KUKA KRL program: MyProgram_327().src

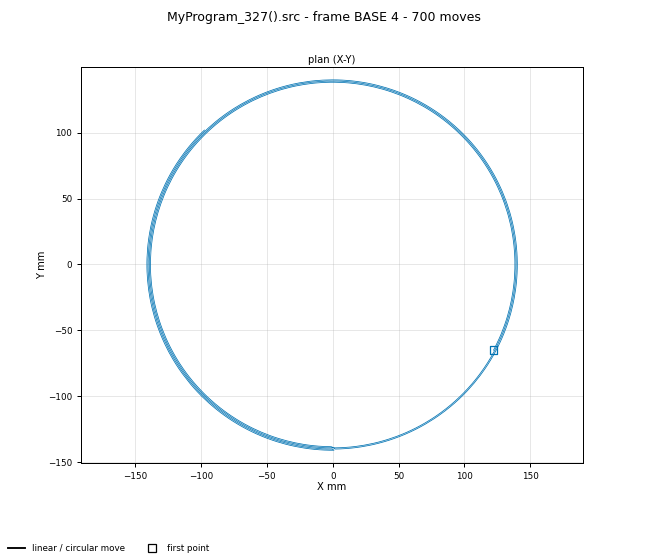
[picture p0: tool path of MyProgram_327().src in frame BASE 4, 700 of 700 moves have a stored position in this frame; points joined in program order, loops and branches not executed]
&ACCESS RVP
&REL 1
&PARAM TEMPLATE = C:\KRC\Roboter\Template\vorgabe
&PARAM EDITMASK = *
DEF MyProgram_327()
; ---- Setting reference (Base) ----
$BASE = BASE_DATA[4]

; --------------------------
; ---- Setting tool (TCP) ----
$TOOL = TOOL_DATA[3]
; --------------------------

$VEL.CP = VEL_APROX_PRINT
Startdeposition()
$VEL.CP = VEL_PRINT
LIN {X 122.1001,Y -65.1036,Z 187,A -22.8126,B 2.4164,C 0.2067,E1 2.5678,E2 476.0313} C_DIS
LIN {X 123.7198,Y -61.9701,Z 187,A -21.3071,B 2.4167,C 0.2026,E1 2.5697,E2 474.5187} C_DIS
LIN {X 125.4053,Y -58.4798,Z 187,A -19.8742,B 2.417,C 0.2,E1 2.5714,E2 473.1074} C_DIS
LIN {X 126.6756,Y -55.679,Z 187,A -18.6979,B 2.4172,C 0.1975,E1 2.5727,E2 471.9431} C_DIS
LIN {X 128.0646,Y -52.404,Z 187,A -17.2,B 2.4175,C 0.1934,E1 2.5743,E2 470.4408} C_DIS
LIN {X 129.3229,Y -49.2171,Z 187,A -15.9923,B 2.4177,C 0.1914,E1 2.5755,E2 469.2602} C_DIS
LIN {X 130.4667,Y -46.1012,Z 187,A -14.659,B 2.4179,C 0.1881,E1 2.5768,E2 467.9313} C_DIS
LIN {X 131.5504,Y -42.9116,Z 187,A -13.3395,B 2.4182,C 0.185,E1 2.5779,E2 466.6208} C_DIS
LIN {X 132.6605,Y -39.3399,Z 187,A -11.9013,B 2.4184,C 0.1818,E1 2.5791,E2 465.1961} C_DIS
LIN {X 133.607,Y -35.9933,Z 187,A -10.6668,B 2.4186,C 0.1796,E1 2.58,E2 463.9876} C_DIS
LIN {X 134.3292,Y -33.2047,Z 187,A -9.3124,B 2.4189,C 0.175,E1 2.5809,E2 462.6111} C_DIS
LIN {X 135.0798,Y -30.0064,Z 187,A -8.0933,B 2.4191,C 0.1724,E1 2.5817,E2 461.4097} C_DIS
LIN {X 135.7603,Y -26.7586,Z 187,A -6.8145,B 2.4193,C 0.1695,E1 2.5824,E2 460.1425} C_DIS
LIN {X 136.44,Y -23.0315,Z 187,A -5.513,B 2.4194,C 0.1674,E1 2.583,E2 458.875} C_DIS
LIN {X 136.8645,Y -20.3723,Z 187,A -4.2723,B 2.4197,C 0.1632,E1 2.5835,E2 457.6172} C_DIS
LIN {X 137.3012,Y -17.1844,Z 187,A -3.0154,B 2.4199,C 0.1602,E1 2.584,E2 456.3692} C_DIS
LIN {X 137.6611,Y -14.0125,Z 187,A -1.7682,B 2.4201,C 0.1571,E1 2.5844,E2 455.1309} C_DIS
LIN {X 137.9882,Y -10.2764,Z 187,A -0.3069,B 2.4204,C 0.1535,E1 2.5847,E2 453.6806} C_DIS
LIN {X 138.2359,Y -6.1423,Z 187,A 1.3133,B 2.4206,C 0.1495,E1 2.5849,E2 452.0716} C_DIS
LIN {X 138.3383,Y -3.0713,Z 187,A 2.5305,B 2.4208,C 0.1464,E1 2.585,E2 450.8609} C_DIS
LIN {X 138.3721,Y 0,Z 187,A 3.7049,B 2.421,C 0.1437,E1 2.585,E2 449.6983} C_DIS
LIN {X 138.3383,Y 3.0713,Z 187,A 5.0506,B 2.4212,C 0.1395,E1 2.585,E2 448.3422} C_DIS
LIN {X 138.1565,Y 7.7265,Z 187,A 6.7524,B 2.4214,C 0.136,E1 2.5847,E2 446.6689} C_DIS
LIN {X 137.9434,Y 10.8859,Z 187,A 8.0939,B 2.4216,C 0.1321,E1 2.5845,E2 445.3227} C_DIS
LIN {X 137.6582,Y 14.0395,Z 187,A 9.2261,B 2.4217,C 0.13,E1 2.5842,E2 444.213} C_DIS
LIN {X 137.2977,Y 17.2115,Z 187,A 10.4775,B 2.4219,C 0.1269,E1 2.5838,E2 442.97} C_DIS
LIN {X 136.8603,Y 20.3995,Z 187,A 11.7392,B 2.4221,C 0.1238,E1 2.5833,E2 441.7166} C_DIS
LIN {X 136.3447,Y 23.601,Z 187,A 13.0011,B 2.4222,C 0.1207,E1 2.5827,E2 440.4644} C_DIS
LIN {X 135.7551,Y 26.786,Z 187,A 14.2905,B 2.4224,C 0.1175,E1 2.582,E2 439.181} C_DIS
LIN {X 135.0798,Y 30.0064,Z 187,A 15.6961,B 2.4226,C 0.1134,E1 2.5812,E2 437.7692} C_DIS
LIN {X 134.1907,Y 33.7517,Z 187,A 17.0979,B 2.4227,C 0.1106,E1 2.5802,E2 436.3913} C_DIS
LIN {X 133.4748,Y 36.4878,Z 187,A 18.1916,B 2.4228,C 0.1081,E1 2.5795,E2 435.307} C_DIS
LIN {X 132.5503,Y 39.7152,Z 187,A 19.5791,B 2.423,C 0.1043,E1 2.5784,E2 433.9191} C_DIS
LIN {X 131.4456,Y 43.2265,Z 187,A 20.9447,B 2.423,C 0.1016,E1 2.5772,E2 432.5732} C_DIS
LIN {X 130.366,Y 46.3814,Z 187,A 22.1708,B 2.4232,C 0.0992,E1 2.5761,E2 431.3662} C_DIS
LIN {X 129.2679,Y 49.3627,Z 187,A 23.5123,B 2.4233,C 0.0955,E1 2.5748,E2 430.0209} C_DIS
LIN {X 127.8426,Y 52.9399,Z 187,A 25.0213,B 2.4235,C 0.092,E1 2.5732,E2 428.522} C_DIS
LIN {X 126.4516,Y 56.1808,Z 187,A 26.2465,B 2.4235,C 0.0902,E1 2.5719,E2 427.3262} C_DIS
LIN {X 125.2281,Y 58.863,Z 187,A 27.5721,B 2.4237,C 0.0861,E1 2.5703,E2 425.9869} C_DIS
LIN {X 123.6932,Y 62.0232,Z 187,A 29.0699,B 2.4238,C 0.0821,E1 2.5684,E2 424.4831} C_DIS
LIN {X 121.6853,Y 65.8758,Z 187,A 30.6655,B 2.4239,C 0.0792,E1 2.5664,E2 422.9127} C_DIS
LIN {X 119.9657,Y 68.9575,Z 187,A 32.0559,B 2.424,C 0.0762,E1 2.5645,E2 421.5308} C_DIS
LIN {X 117.854,Y 72.5066,Z 187,A 33.7517,B 2.4242,C 0.0721,E1 2.562,E2 419.8363} C_DIS
LIN {X 115.8171,Y 75.7187,Z 187,A 35.1883,B 2.4242,C 0.0694,E1 2.5599,E2 418.4167} C_DIS
LIN {X 113.8287,Y 78.6762,Z 187,A 36.5912,B 2.4243,C 0.0665,E1 2.5577,E2 417.0225} C_DIS
LIN {X 111.4897,Y 81.9559,Z 187,A 38.2376,B 2.4244,C 0.0628,E1 2.555,E2 415.3784} C_DIS
LIN {X 109.0842,Y 85.1325,Z 187,A 39.7581,B 2.4244,C 0.06,E1 2.5524,E2 413.8739} C_DIS
LIN {X 106.8509,Y 87.9193,Z 187,A 41.1713,B 2.4245,C 0.0572,E1 2.55,E2 412.4686} C_DIS
LIN {X 104.2126,Y 91.03,Z 187,A 42.8402,B 2.4246,C 0.0537,E1 2.5469,E2 410.8019} C_DIS
LIN {X 101.5684,Y 93.9722,Z 187,A 44.3542,B 2.4246,C 0.0511,E1 2.5441,E2 409.3031} C_DIS
LIN {X 98.7051,Y 96.9744,Z 187,A 46.0508,B 2.4248,C 0.0477,E1 2.5408,E2 407.6089} C_DIS
LIN {X 95.915,Y 99.7357,Z 187,A 47.5589,B 2.4248,C 0.0452,E1 2.5378,E2 406.1153} C_DIS
LIN {X 93.3132,Y 102.1742,Z 187,A 48.9762,B 2.4248,C 0.0427,E1 2.5349,E2 404.7052} C_DIS
LIN {X 90.2523,Y 104.8869,Z 187,A 50.655,B 2.4249,C 0.0396,E1 2.5314,E2 403.0281} C_DIS
LIN {X 87.2159,Y 107.4259,Z 187,A 52.1798,B 2.4249,C 0.0373,E1 2.5281,E2 401.5174} C_DIS
LIN {X 83.9895,Y 109.9659,Z 187,A 53.8641,B 2.4249,C 0.0344,E1 2.5244,E2 399.835} C_DIS
LIN {X 80.6649,Y 112.4275,Z 187,A 55.4338,B 2.425,C 0.0324,E1 2.5209,E2 398.283} C_DIS
LIN {X 77.9316,Y 114.3398,Z 187,A 56.8056,B 2.425,C 0.0301,E1 2.5177,E2 396.9124} C_DIS
LIN {X 74.9631,Y 116.3075,Z 187,A 58.222,B 2.425,C 0.0281,E1 2.5144,E2 395.5032} C_DIS
LIN {X 71.9662,Y 118.1854,Z 187,A 59.6383,B 2.425,C 0.0261,E1 2.5111,E2 394.0929} C_DIS
LIN {X 68.9446,Y 119.9732,Z 187,A 61.0497,B 2.4251,C 0.0241,E1 2.5077,E2 392.6868} C_DIS
LIN {X 65.8626,Y 121.6923,Z 187,A 62.5626,B 2.4251,C 0.0216,E1 2.504,E2 391.1677} C_DIS
LIN {X 63.1849,Y 123.1018,Z 187,A 63.5476,B 2.4251,C 0.0216,E1 2.5016,E2 390.2156} C_DIS
LIN {X 60.4063,Y 124.4908,Z 187,A 64.9206,B 2.4251,C 0.0193,E1 2.4981,E2 388.8323} C_DIS
LIN {X 57.2872,Y 125.9567,Z 187,A 66.4596,B 2.4251,C 0.0167,E1 2.4942,E2 387.2797} C_DIS
LIN {X 54.0928,Y 127.3611,Z 187,A 67.7144,B 2.4251,C 0.0162,E1 2.491,E2 386.0484} C_DIS
LIN {X 50.9342,Y 128.6571,Z 187,A 69.113,B 2.4251,C 0.0146,E1 2.4874,E2 384.6519} C_DIS
LIN {X 47.6023,Y 129.9258,Z 187,A 70.6471,B 2.4251,C 0.0125,E1 2.4834,E2 383.111} C_DIS
LIN {X 44.4938,Y 131.0236,Z 187,A 71.8665,B 2.4251,C 0.012,E1 2.4802,E2 381.9097} C_DIS
LIN {X 41.3004,Y 132.0652,Z 187,A 73.348,B 2.4252,C 0.0101,E1 2.4762,E2 380.4175} C_DIS
LIN {X 37.9383,Y 133.0691,Z 187,A 74.7459,B 2.4252,C 0.009,E1 2.4725,E2 379.0265} C_DIS
LIN {X 34.4003,Y 134.0261,Z 187,A 76.0725,B 2.4252,C 0.0089,E1 2.4689,E2 377.7236} C_DIS
LIN {X 31.5914,Y 134.7177,Z 187,A 77.3145,B 2.4252,C 0.0077,E1 2.4655,E2 376.4766} C_DIS
LIN {X 28.368,Y 135.4332,Z 187,A 78.6682,B 2.4252,C 0.0067,E1 2.4619,E2 375.125} C_DIS
LIN {X 25.1787,Y 136.0623,Z 187,A 80.1111,B 2.4252,C 0.0052,E1 2.4579,E2 373.6707} C_DIS
LIN {X 21.7901,Y 136.645,Z 187,A 81.3295,B 2.4252,C 0.0055,E1 2.4546,E2 372.4777} C_DIS
LIN {X 18.5226,Y 137.1258,Z 187,A 82.6526,B 2.4252,C 0.005,E1 2.4509,E2 371.1604} C_DIS
LIN {X 15.5963,Y 137.4907,Z 187,A 83.9522,B 2.4252,C 0.004,E1 2.4473,E2 369.8518} C_DIS
LIN {X 12.4334,Y 137.8127,Z 187,A 85.3941,B 2.4252,C 0.0027,E1 2.4432,E2 368.395} C_DIS
LIN {X 7.7,Y 138.1579,Z 187,A 87.2012,B 2.4252,C 0.0029,E1 2.4382,E2 366.6079} C_DIS
LIN {X 4.5906,Y 138.2961,Z 187,A 88.4803,B 2.4252,C 0.0026,E1 2.4347,E2 365.3305} C_DIS
LIN {X 1.5062,Y 138.3641,Z 187,A 89.74,B 2.4252,C 0.0024,E1 2.4311,E2 364.0734} C_DIS
LIN {X -1.5323,Y 138.3639,Z 187,A 91.159,B 2.4252,C 0.0014,E1 2.4271,E2 362.6355} C_DIS
LIN {X -6.1687,Y 138.2348,Z 187,A 93.0324,B 2.4252,C 0.0015,E1 2.4219,E2 360.7686} C_DIS
LIN {X -9.3168,Y 138.0583,Z 187,A 94.2351,B 2.4252,C 0.0021,E1 2.4186,E2 359.579} C_DIS
LIN {X -12.4603,Y 137.8101,Z 187,A 95.5449,B 2.4252,C 0.0021,E1 2.4149,E2 358.2693} C_DIS
LIN {X -15.6233,Y 137.4874,Z 187,A 96.868,B 2.4252,C 0.0023,E1 2.4112,E2 356.946} C_DIS
LIN {X -19.3499,Y 137.0106,Z 187,A 98.2332,B 2.4252,C 0.0035,E1 2.4075,E2 355.6045} C_DIS
LIN {X -21.9988,Y 136.6124,Z 187,A 99.5506,B 2.4252,C 0.0028,E1 2.4038,E2 354.2626} C_DIS
LIN {X -25.1787,Y 136.0623,Z 187,A 100.8981,B 2.4252,C 0.0032,E1 2.4001,E2 352.9144} C_DIS
LIN {X -28.4228,Y 135.4217,Z 187,A 102.2713,B 2.4252,C 0.0037,E1 2.3963,E2 351.5415} C_DIS
LIN {X -32.0101,Y 134.6172,Z 187,A 103.8238,B 2.4252,C 0.0043,E1 2.3921,E2 349.9861} C_DIS
LIN {X -35.4295,Y 133.7574,Z 187,A 105.0908,B 2.4252,C 0.006,E1 2.3887,E2 348.7433} C_DIS
LIN {X -38.1018,Y 133.0231,Z 187,A 106.465,B 2.4252,C 0.0056,E1 2.3849,E2 347.3423} C_DIS
LIN {X -41.3278,Y 132.0564,Z 187,A 107.9329,B 2.4252,C 0.0063,E1 2.381,E2 345.8662} C_DIS
LIN {X -44.9938,Y 130.8506,Z 187,A 109.3186,B 2.4252,C 0.0084,E1 2.3774,E2 344.5071} C_DIS
LIN {X -47.7335,Y 129.8786,Z 187,A 110.7439,B 2.4252,C 0.0084,E1 2.3736,E2 343.0557} C_DIS
LIN {X -50.9613,Y 128.6461,Z 187,A 112.1811,B 2.4252,C 0.0096,E1 2.3698,E2 341.6187} C_DIS
LIN {X -54.1198,Y 127.3498,Z 187,A 113.6472,B 2.4252,C 0.0107,E1 2.366,E2 340.147} C_DIS
LIN {X -57.5131,Y 125.8523,Z 187,A 115.1129,B 2.4252,C 0.0126,E1 2.3623,E2 338.6908} C_DIS
LIN {X -60.433,Y 124.478,Z 187,A 116.5871,B 2.4252,C 0.0134,E1 2.3585,E2 337.2007} C_DIS
LIN {X -63.5801,Y 122.9001,Z 187,A 118.0597,B 2.4252,C 0.0151,E1 2.3549,E2 335.7272} C_DIS
LIN {X -67.1845,Y 120.967,Z 187,A 119.8497,B 2.4252,C 0.0167,E1 2.3504,E2 333.9265} C_DIS
LIN {X -71.0089,Y 118.7624,Z 187,A 121.7285,B 2.4252,C 0.0189,E1 2.3459,E2 332.0427} C_DIS
LIN {X -74.2303,Y 116.7766,Z 187,A 123.3063,B 2.4252,C 0.021,E1 2.3422,E2 330.4647} C_DIS
LIN {X -77.2092,Y 114.8288,Z 187,A 124.8272,B 2.4252,C 0.023,E1 2.3386,E2 328.939} C_DIS
LIN {X -80.2682,Y 112.7112,Z 187,A 126.3729,B 2.4251,C 0.0253,E1 2.3351,E2 327.3937} C_DIS
LIN {X -82.9959,Y 110.7186,Z 187,A 127.8659,B 2.4251,C 0.0271,E1 2.3317,E2 325.8901} C_DIS
LIN {X -85.8342,Y 108.533,Z 187,A 129.4028,B 2.4251,C 0.0294,E1 2.3283,E2 324.3478} C_DIS
LIN {X -88.6075,Y 106.2809,Z 187,A 130.9371,B 2.4251,C 0.0317,E1 2.325,E2 322.8077} C_DIS
LIN {X -91.4291,Y 103.863,Z 187,A 132.4964,B 2.425,C 0.0343,E1 2.3217,E2 321.247} C_DIS
LIN {X -93.9722,Y 101.5684,Z 187,A 134.01,B 2.425,C 0.0366,E1 2.3185,E2 319.7227} C_DIS
LIN {X -96.9482,Y 98.7308,Z 187,A 135.8359,B 2.425,C 0.0394,E1 2.3148,E2 317.8829} C_DIS
LIN {X -99.7357,Y 95.915,Z 187,A 137.6067,B 2.4249,C 0.0421,E1 2.3113,E2 316.0971} C_DIS
LIN {X -102.7757,Y 92.6504,Z 187,A 139.4216,B 2.4248,C 0.0459,E1 2.3079,E2 314.2875} C_DIS
LIN {X -105.1371,Y 89.9618,Z 187,A 140.9701,B 2.4248,C 0.0488,E1 2.3051,E2 312.7319} C_DIS
LIN {X -107.4259,Y 87.2159,Z 187,A 142.5188,B 2.4247,C 0.0517,E1 2.3023,E2 311.1758} C_DIS
LIN {X -109.9373,Y 84.0268,Z 187,A 144.34,B 2.4247,C 0.0549,E1 2.2992,E2 309.3384} C_DIS
LIN {X -112.3001,Y 80.8432,Z 187,A 146.0009,B 2.4245,C 0.0585,E1 2.2964,E2 307.6763} C_DIS
LIN {X -114.3398,Y 77.9316,Z 187,A 147.5506,B 2.4245,C 0.0616,E1 2.2939,E2 306.118} C_DIS
LIN {X -116.3075,Y 74.9631,Z 187,A 149.091,B 2.4244,C 0.0648,E1 2.2916,E2 304.5706} C_DIS
LIN {X -118.4844,Y 71.4716,Z 187,A 150.9272,B 2.4243,C 0.0685,E1 2.2889,E2 302.7191} C_DIS
LIN {X -120.4164,Y 68.1674,Z 187,A 152.5555,B 2.4242,C 0.0722,E1 2.2866,E2 301.0865} C_DIS
LIN {X -122.1001,Y 65.1036,Z 187,A 154.0804,B 2.424,C 0.0755,E1 2.2846,E2 299.5531} C_DIS
LIN {X -123.9238,Y 61.5565,Z 187,A 155.7873,B 2.424,C 0.0794,E1 2.2824,E2 297.8403} C_DIS
LIN {X -125.2281,Y 58.863,Z 187,A 157.1291,B 2.4238,C 0.0823,E1 2.2808,E2 296.4867} C_DIS
LIN {X -126.6756,Y 55.679,Z 187,A 158.658,B 2.4238,C 0.0858,E1 2.279,E2 294.9487} C_DIS
LIN {X -128.0141,Y 52.5291,Z 187,A 160.3126,B 2.4236,C 0.0889,E1 2.2772,E2 293.2653} C_DIS
LIN {X -129.4826,Y 48.7907,Z 187,A 161.7021,B 2.4234,C 0.0938,E1 2.2759,E2 291.9113} C_DIS
LIN {X -130.4667,Y 46.1012,Z 187,A 163.1671,B 2.4234,C 0.0963,E1 2.2744,E2 290.4122} C_DIS
LIN {X -131.5504,Y 42.9116,Z 187,A 164.7514,B 2.4232,C 0.0995,E1 2.273,E2 288.8048} C_DIS
LIN {X -132.5587,Y 39.6878,Z 187,A 166.1236,B 2.423,C 0.1034,E1 2.2719,E2 287.437} C_DIS
LIN {X -133.6118,Y 35.9752,Z 187,A 167.8218,B 2.4228,C 0.1074,E1 2.2706,E2 285.7272} C_DIS
LIN {X -134.389,Y 32.9567,Z 187,A 169.0851,B 2.4227,C 0.111,E1 2.2698,E2 284.4682} C_DIS
LIN {X -135.0798,Y 30.0064,Z 187,A 170.5235,B 2.4225,C 0.114,E1 2.2689,E2 283.0074} C_DIS
LIN {X -135.7603,Y 26.7586,Z 187,A 171.9589,B 2.4224,C 0.1176,E1 2.2681,E2 281.5652} C_DIS
LIN {X -136.4308,Y 23.087,Z 187,A 173.6218,B 2.4222,C 0.1217,E1 2.2673,E2 279.8883} C_DIS
LIN {X -136.8645,Y 20.3723,Z 187,A 174.8153,B 2.422,C 0.1247,E1 2.2668,E2 278.6886} C_DIS
LIN {X -137.3012,Y 17.1844,Z 187,A 176.2283,B 2.4218,C 0.1282,E1 2.2662,E2 277.2661} C_DIS
LIN {X -137.6611,Y 14.0125,Z 187,A 177.7952,B 2.4217,C 0.1313,E1 2.2658,E2 275.6687} C_DIS
LIN {X -137.9971,Y 10.1551,Z 187,A 179.3602,B 2.4214,C 0.1359,E1 2.2654,E2 274.1096} C_DIS
LIN {X -138.2359,Y 6.1423,Z 187,A -178.9025,B 2.4212,C 0.1404,E1 2.2652,E2 272.364} C_DIS
LIN {X -138.3388,Y 3.0451,Z 187,A -177.5311,B 2.421,C 0.1438,E1 2.2651,E2 270.9821} C_DIS
LIN {X -138.3721,Y 0,Z 187,A -176.2115,B 2.4208,C 0.1472,E1 2.2651,E2 269.6558} C_DIS
LIN {X -138.3234,Y -3.6077,Z 187,A -174.6047,B 2.4205,C 0.1512,E1 2.2651,E2 268.0352} C_DIS
LIN {X -138.1565,Y -7.7265,Z 187,A -172.7823,B 2.4202,C 0.1557,E1 2.2654,E2 266.199} C_DIS
LIN {X -137.9148,Y -11.2245,Z 187,A -171.3766,B 2.42,C 0.1599,E1 2.2657,E2 264.8001} C_DIS
LIN {X -137.6582,Y -14.0395,Z 187,A -170.0002,B 2.4198,C 0.1626,E1 2.266,E2 263.3977} C_DIS
LIN {X -137.2684,Y -17.4343,Z 187,A -168.4258,B 2.4195,C 0.1662,E1 2.2666,E2 261.8032} C_DIS
LIN {X -136.7861,Y -20.879,Z 187,A -167.1476,B 2.4192,C 0.1706,E1 2.2671,E2 260.547} C_DIS
LIN {X -136.3447,Y -23.601,Z 187,A -165.7581,B 2.419,C 0.1731,E1 2.2677,E2 259.1259} C_DIS
LIN {X -135.7551,Y -26.786,Z 187,A -164.2167,B 2.4188,C 0.1763,E1 2.2686,E2 257.559} C_DIS
LIN {X -134.9919,Y -30.3909,Z 187,A -162.673,B 2.4185,C 0.1805,E1 2.2695,E2 256.0137} C_DIS
LIN {X -134.1798,Y -33.7948,Z 187,A -161.3875,B 2.4182,C 0.1848,E1 2.2703,E2 254.7503} C_DIS
LIN {X -133.4748,Y -36.4878,Z 187,A -159.9345,B 2.418,C 0.1872,E1 2.2714,E2 253.2586} C_DIS
LIN {X -132.5445,Y -39.7341,Z 187,A -158.4602,B 2.4177,C 0.1907,E1 2.2725,E2 251.775} C_DIS
LIN {X -131.5504,Y -42.9116,Z 187,A -156.9903,B 2.4174,C 0.1941,E1 2.2738,E2 250.2937} C_DIS
LIN {X -130.4572,Y -46.1286,Z 187,A -155.4993,B 2.4172,C 0.1976,E1 2.2752,E2 248.7923} C_DIS
LIN {X -129.2679,Y -49.3627,Z 187,A -153.9878,B 2.4169,C 0.2011,E1 2.2767,E2 247.2702} C_DIS
LIN {X -127.8703,Y -52.8734,Z 187,A -152.477,B 2.4165,C 0.2052,E1 2.2783,E2 245.7671} C_DIS
LIN {X -126.6519,Y -55.733,Z 187,A -150.9705,B 2.4163,C 0.2079,E1 2.28,E2 244.2321} C_DIS
LIN {X -125.2281,Y -58.863,Z 187,A -149.3668,B 2.416,C 0.211,E1 2.2819,E2 242.6051} C_DIS
LIN {X -123.5919,Y -62.2222,Z 187,A -147.9172,B 2.4157,C 0.215,E1 2.2836,E2 241.169} C_DIS
LIN {X -121.9816,Y -65.3243,Z 187,A -146.1969,B 2.4154,C 0.2178,E1 2.2859,E2 239.4129} C_DIS
LIN {X -119.9657,Y -68.9575,Z 187,A -144.4926,B 2.4151,C 0.2219,E1 2.2883,E2 237.7113} C_DIS
LIN {X -117.9062,Y -72.4215,Z 187,A -142.683,B 2.4147,C 0.2254,E1 2.2909,E2 235.8834} C_DIS
LIN {X -115.8171,Y -75.7187,Z 187,A -141.0326,B 2.4144,C 0.229,E1 2.2934,E2 234.2289} C_DIS
LIN {X -113.525,Y -79.1126,Z 187,A -139.2026,B 2.4141,C 0.2324,E1 2.2963,E2 232.3813} C_DIS
LIN {X -111.2506,Y -82.2814,Z 187,A -137.5621,B 2.4137,C 0.2358,E1 2.299,E2 230.7379} C_DIS
LIN {X -109.0842,Y -85.1325,Z 187,A -135.8993,B 2.4135,C 0.2384,E1 2.3019,E2 229.0511} C_DIS
LIN {X -106.2809,Y -88.6075,Z 187,A -133.9897,B 2.4131,C 0.2421,E1 2.3053,E2 227.1338} C_DIS
LIN {X -103.3625,Y -91.9951,Z 187,A -132.1455,B 2.4127,C 0.2458,E1 2.3087,E2 225.2909} C_DIS
LIN {X -100.9583,Y -94.6274,Z 187,A -130.4891,B 2.4125,C 0.2481,E1 2.3119,E2 223.6103} C_DIS
LIN {X -97.8441,Y -97.8441,Z 187,A -128.6707,B 2.4121,C 0.2517,E1 2.3155,E2 221.7969} C_DIS
LIN {X -95.2676,Y -100.3543,Z 187,A -127.1216,B 2.4119,C 0.2542,E1 2.3186,E2 220.24} C_DIS
LIN {X -92.2748,Y -103.1121,Z 187,A -125.3125,B 2.4116,C 0.2567,E1 2.3224,E2 218.4142} C_DIS
LIN {X -89.2806,Y -105.7161,Z 187,A -123.6682,B 2.4113,C 0.2595,E1 2.3259,E2 216.7698} C_DIS
LIN {X -86.0952,Y -108.3252,Z 187,A -121.8458,B 2.4111,C 0.2618,E1 2.3299,E2 214.9315} C_DIS
LIN {X -82.9837,Y -110.7277,Z 187,A -120.2208,B 2.4108,C 0.2644,E1 2.3335,E2 213.307} C_DIS
LIN {X -80.1196,Y -112.8174,Z 187,A -118.7013,B 2.4106,C 0.2663,E1 2.337,E2 211.7805} C_DIS
LIN {X -76.7228,Y -115.1536,Z 187,A -116.8993,B 2.4103,C 0.2684,E1 2.3412,E2 209.9655} C_DIS
LIN {X -73.4823,Y -117.2488,Z 187,A -115.299,B 2.4101,C 0.2705,E1 2.3449,E2 208.3648} C_DIS
LIN {X -70.4591,Y -119.09,Z 187,A -113.8003,B 2.4099,C 0.2723,E1 2.3486,E2 206.8614} C_DIS
LIN {X -66.9138,Y -121.1169,Z 187,A -112.0227,B 2.4097,C 0.274,E1 2.3529,E2 205.0719} C_DIS
LIN {X -63.5537,Y -122.914,Z 187,A -110.4381,B 2.4095,C 0.2757,E1 2.3568,E2 203.4861} C_DIS
LIN {X -60.4063,Y -124.4908,Z 187,A -108.8193,B 2.4095,C 0.2765,E1 2.361,E2 201.8451} C_DIS
LIN {X -57.135,Y -126.0248,Z 187,A -107.4828,B 2.4092,C 0.2788,E1 2.3643,E2 200.5302} C_DIS
LIN {X -54.0928,Y -127.3611,Z 187,A -106.0417,B 2.409,C 0.2797,E1 2.368,E2 199.0799} C_DIS
LIN {X -50.4991,Y -128.8262,Z 187,A -104.4609,B 2.4089,C 0.2813,E1 2.3721,E2 197.5023} C_DIS
LIN {X -47.7062,Y -129.8884,Z 187,A -103.139,B 2.4089,C 0.2818,E1 2.3756,E2 196.1686} C_DIS
LIN {X -44.4938,Y -131.0236,Z 187,A -101.7189,B 2.4087,C 0.2828,E1 2.3794,E2 194.7469} C_DIS
LIN {X -40.9901,Y -132.1601,Z 187,A -100.0974,B 2.4087,C 0.2833,E1 2.3837,E2 193.1118} C_DIS
LIN {X -37.547,Y -133.1786,Z 187,A -98.7453,B 2.4084,C 0.2849,E1 2.3873,E2 191.7776} C_DIS
LIN {X -34.8186,Y -133.9199,Z 187,A -97.4786,B 2.4084,C 0.285,E1 2.3908,E2 190.4975} C_DIS
LIN {X -31.5914,Y -134.7177,Z 187,A -96.1006,B 2.4084,C 0.2856,E1 2.3945,E2 189.1189} C_DIS
LIN {X -28.368,Y -135.4332,Z 187,A -94.5722,B 2.4084,C 0.2853,E1 2.3988,E2 187.5679} C_DIS
LIN {X -25.1787,Y -136.0623,Z 187,A -93.3609,B 2.4083,C 0.2865,E1 2.4021,E2 186.3747} C_DIS
LIN {X -21.9715,Y -136.6169,Z 187,A -92.0081,B 2.4083,C 0.2868,E1 2.4058,E2 185.0207} C_DIS
LIN {X -18.7765,Y -137.0926,Z 187,A -90.6672,B 2.4082,C 0.287,E1 2.4095,E2 183.6788} C_DIS
LIN {X -15.191,Y -137.5343,Z 187,A -89.1129,B 2.4082,C 0.2869,E1 2.4139,E2 182.1157} C_DIS
LIN {X -10.8591,Y -137.9457,Z 187,A -87.3605,B 2.4082,C 0.2872,E1 2.4187,E2 180.3695} C_DIS
LIN {X -7.7,Y -138.1579,Z 187,A -86.0624,B 2.4082,C 0.2872,E1 2.4224,E2 179.0726} C_DIS
LIN {X -4.5906,Y -138.2961,Z 187,A -84.7785,B 2.4082,C 0.2872,E1 2.4259,E2 177.7887} C_DIS
LIN {X -1.1044,Y -138.3663,Z 187,A -83.2901,B 2.4082,C 0.2867,E1 2.4301,E2 176.2935} C_DIS
LIN {X -1.1044,Y -138.3663,Z 187,A -83.2901,B 2.4082,C 0.2867,E1 2.4301,E2 176.2935} C_DIS
Enddeposition()
LIN {X 0.9877,Y -139.2619,Z 187,A -82.7944,B 2.4115,C 0.2901,E1 2.435,E2 175.8768} C_DIS
Startdeposition()
$VEL.CP = VEL_PRINT
LIN {X -2.3088,Y -139.2508,Z 187,A -84.4091,B 2.4113,C 0.2919,E1 2.4304,E2 177.5278} C_DIS
LIN {X -5.5487,Y -139.1594,Z 187,A -85.7032,B 2.4113,C 0.2919,E1 2.4267,E2 178.8172} C_DIS
LIN {X -9.2772,Y -138.9624,Z 187,A -87.2347,B 2.4113,C 0.2919,E1 2.4225,E2 180.3487} C_DIS
LIN {X -12.6549,Y -138.6952,Z 187,A -88.7627,B 2.4113,C 0.2926,E1 2.4182,E2 181.8957} C_DIS
LIN {X -16.6138,Y -138.2753,Z 187,A -90.3124,B 2.4113,C 0.2919,E1 2.4139,E2 183.4339} C_DIS
LIN {X -19.9208,Y -137.8379,Z 187,A -91.6625,B 2.4113,C 0.2915,E1 2.4101,E2 184.7816} C_DIS
LIN {X -23.744,Y -137.2331,Z 187,A -93.4296,B 2.4113,C 0.2921,E1 2.4052,E2 186.5732} C_DIS
LIN {X -26.8449,Y -136.6598,Z 187,A -94.7351,B 2.4113,C 0.2917,E1 2.4016,E2 187.8803} C_DIS
LIN {X -34.2357,Y -134.9961,Z 187,A -97.7968,B 2.4115,C 0.29,E1 2.3933,E2 190.9354} C_DIS
LIN {X -37.8207,Y -134.0362,Z 187,A -99.2595,B 2.4117,C 0.2888,E1 2.3894,E2 192.3899} C_DIS
LIN {X -41.1368,Y -133.0561,Z 187,A -100.8433,B 2.4117,C 0.2888,E1 2.3851,E2 193.996} C_DIS
LIN {X -44.6421,Y -131.9225,Z 187,A -102.228,B 2.4119,C 0.2871,E1 2.3814,E2 195.3634} C_DIS
LIN {X -48.4707,Y -130.5631,Z 187,A -103.7872,B 2.4121,C 0.2853,E1 2.3774,E2 196.9075} C_DIS
LIN {X -52.3491,Y -129.0567,Z 187,A -105.774,B 2.4121,C 0.2851,E1 2.3721,E2 198.9323} C_DIS
LIN {X -55.8014,Y -127.6029,Z 187,A -107.5551,B 2.4121,C 0.2848,E1 2.3674,E2 200.7464} C_DIS
LIN {X -60.2863,Y -125.5452,Z 187,A -110.2147,B 2.4121,C 0.2856,E1 2.3605,E2 203.4914} C_DIS
LIN {X -66.0686,Y -122.603,Z 187,A -111.9415,B 2.4129,C 0.2784,E1 2.3565,E2 205.0911} C_DIS
LIN {X -69.0439,Y -120.9523,Z 187,A -113.5949,B 2.4129,C 0.2778,E1 2.3524,E2 206.7791} C_DIS
LIN {X -72.9148,Y -118.659,Z 187,A -115.4727,B 2.4132,C 0.2755,E1 2.3479,E2 208.6607} C_DIS
LIN {X -77.2218,Y -115.9023,Z 187,A -118.7818,B 2.413,C 0.2775,E1 2.3399,E2 212.132} C_DIS
LIN {X -83.8388,Y -111.2096,Z 187,A -120.8626,B 2.4141,C 0.2675,E1 2.3355,E2 214.0439} C_DIS
LIN {X -86.3637,Y -109.2612,Z 187,A -122.5148,B 2.4142,C 0.2667,E1 2.3318,E2 215.7423} C_DIS
LIN {X -89.955,Y -106.3236,Z 187,A -124.4795,B 2.4145,C 0.2637,E1 2.3275,E2 217.7144} C_DIS
LIN {X -93.3528,Y -103.3531,Z 187,A -126.4245,B 2.4149,C 0.2608,E1 2.3234,E2 219.6712} C_DIS
LIN {X -96.6167,Y -100.3089,Z 187,A -128.4764,B 2.4151,C 0.2583,E1 2.3192,E2 221.752} C_DIS
LIN {X -99.4473,Y -97.5025,Z 187,A -129.996,B 2.4155,C 0.2548,E1 2.3163,E2 223.2551} C_DIS
LIN {X -102.5613,Y -94.2215,Z 187,A -132.0057,B 2.4158,C 0.2516,E1 2.3124,E2 225.2846} C_DIS
LIN {X -104.8547,Y -91.6626,Z 187,A -133.3635,B 2.4161,C 0.2486,E1 2.3099,E2 226.6347} C_DIS
LIN {X -107.5554,Y -88.4791,Z 187,A -135.2515,B 2.4164,C 0.2457,E1 2.3065,E2 228.5452} C_DIS
LIN {X -110.2581,Y -85.0868,Z 187,A -137.3965,B 2.4167,C 0.243,E1 2.3027,E2 230.7379} C_DIS
LIN {X -112.5873,Y -81.98,Z 187,A -138.6288,B 2.4172,C 0.2384,E1 2.3008,E2 231.9211} C_DIS
LIN {X -114.7804,Y -78.8795,Z 187,A -140.3883,B 2.4174,C 0.2355,E1 2.2979,E2 233.7066} C_DIS
LIN {X -117.3143,Y -75.0591,Z 187,A -142.5211,B 2.4178,C 0.232,E1 2.2946,E2 235.8717} C_DIS
LIN {X -119.8559,Y -70.9315,Z 187,A -145.138,B 2.4181,C 0.2291,E1 2.2908,E2 238.5702} C_DIS
LIN {X -122.6369,Y -66.0054,Z 187,A -146.8981,B 2.4187,C 0.2219,E1 2.2885,E2 240.2547} C_DIS
LIN {X -124.2911,Y -62.8317,Z 187,A -148.3792,B 2.4191,C 0.2183,E1 2.2866,E2 241.7365} C_DIS
LIN {X -125.8131,Y -59.7255,Z 187,A -149.9262,B 2.4193,C 0.2151,E1 2.2847,E2 243.2993} C_DIS
LIN {X -127.7175,Y -55.5364,Z 187,A -152.0171,B 2.4197,C 0.2109,E1 2.2823,E2 245.4156} C_DIS
LIN {X -128.9754,Y -52.5509,Z 187,A -153.3953,B 2.42,C 0.2076,E1 2.2808,E2 246.7992} C_DIS
LIN {X -131.3155,Y -46.3995,Z 187,A -156.1381,B 2.4206,C 0.2007,E1 2.2782,E2 249.5456} C_DIS
LIN {X -132.372,Y -43.2922,Z 187,A -157.5663,B 2.4209,C 0.1973,E1 2.2769,E2 250.9835} C_DIS
LIN {X -133.1424,Y -40.8548,Z 187,A -158.6933,B 2.4211,C 0.1947,E1 2.2759,E2 252.1197} C_DIS
LIN {X -134.1086,Y -37.5619,Z 187,A -160.1928,B 2.4214,C 0.1912,E1 2.2748,E2 253.63} C_DIS
LIN {X -134.9859,Y -34.2757,Z 187,A -161.6638,B 2.4216,C 0.1876,E1 2.2737,E2 255.1098} C_DIS
LIN {X -135.7936,Y -30.9214,Z 187,A -163.1689,B 2.4219,C 0.1839,E1 2.2728,E2 256.6253} C_DIS
LIN {X -136.4768,Y -27.7509,Z 187,A -164.6087,B 2.4222,C 0.1805,E1 2.2719,E2 258.0782} C_DIS
LIN {X -137.2193,Y -23.8207,Z 187,A -166.596,B 2.4224,C 0.1768,E1 2.2709,E2 260.1091} C_DIS
LIN {X -137.8851,Y -19.5902,Z 187,A -168.1983,B 2.4228,C 0.1716,E1 2.2703,E2 261.6897} C_DIS
LIN {X -138.3802,Y -15.7344,Z 187,A -169.8832,B 2.4231,C 0.1673,E1 2.2697,E2 263.3849} C_DIS
LIN {X -138.7549,Y -11.9679,Z 187,A -171.3295,B 2.4234,C 0.1627,E1 2.2693,E2 264.8158} C_DIS
LIN {X -139.2009,Y -4.4207,Z 187,A -174.8372,B 2.4239,C 0.1549,E1 2.2688,E2 268.3732} C_DIS
LIN {X -139.2454,Y 2.6364,Z 187,A -177.9217,B 2.4244,C 0.1472,E1 2.2688,E2 271.4793} C_DIS
LIN {X -138.9713,Y 9.1325,Z 187,A 179.268,B 2.4249,C 0.14,E1 2.2691,E2 274.3054} C_DIS
LIN {X -138.7587,Y 11.9228,Z 187,A 177.965,B 2.425,C 0.1371,E1 2.2694,E2 275.627} C_DIS
LIN {X -138.4008,Y 15.5476,Z 187,A 175.9614,B 2.4252,C 0.1341,E1 2.2701,E2 277.6939} C_DIS
LIN {X -137.9259,Y 19.3048,Z 187,A 174.5104,B 2.4254,C 0.1295,E1 2.2706,E2 279.1304} C_DIS
LIN {X -137.1876,Y 23.9982,Z 187,A 172.5173,B 2.4257,C 0.1242,E1 2.2715,E2 281.127} C_DIS
LIN {X -136.2965,Y 28.633,Z 187,A 170.6261,B 2.426,C 0.1187,E1 2.2725,E2 283.0105} C_DIS
LIN {X -135.6232,Y 31.6674,Z 187,A 169.2713,B 2.4261,C 0.1154,E1 2.2734,E2 284.3741} C_DIS
LIN {X -134.9509,Y 34.4136,Z 187,A 167.9822,B 2.4263,C 0.1125,E1 2.2743,E2 285.6782} C_DIS
LIN {X -133.9407,Y 38.1624,Z 187,A 166.3099,B 2.4265,C 0.1084,E1 2.2755,E2 287.359} C_DIS
LIN {X -133.1295,Y 40.8968,Z 187,A 165.0627,B 2.4266,C 0.1054,E1 2.2765,E2 288.6145} C_DIS
LIN {X -132.0247,Y 44.335,Z 187,A 163.403,B 2.4268,C 0.1019,E1 2.278,E2 290.2951} C_DIS
LIN {X -130.8908,Y 47.5787,Z 187,A 161.9746,B 2.4269,C 0.0982,E1 2.2793,E2 291.7243} C_DIS
LIN {X -129.672,Y 50.8065,Z 187,A 160.4737,B 2.427,C 0.0947,E1 2.2809,E2 293.2344} C_DIS
LIN {X -128.1741,Y 54.4796,Z 187,A 158.7684,B 2.4272,C 0.0907,E1 2.2827,E2 294.9478} C_DIS
LIN {X -127.1012,Y 56.9321,Z 187,A 157.5859,B 2.4272,C 0.088,E1 2.284,E2 296.1395} C_DIS
LIN {X -125.5195,Y 60.3401,Z 187,A 155.9463,B 2.4274,C 0.0844,E1 2.286,E2 297.7898} C_DIS
LIN {X -123.871,Y 63.6569,Z 187,A 154.3586,B 2.4275,C 0.0808,E1 2.288,E2 299.3844} C_DIS
LIN {X -122.1361,Y 66.9282,Z 187,A 152.6836,B 2.4277,C 0.0775,E1 2.2903,E2 301.0772} C_DIS
LIN {X -119.1976,Y 72.0309,Z 187,A 150.3016,B 2.4278,C 0.0716,E1 2.2936,E2 303.4524} C_DIS
LIN {X -115.999,Y 77.0769,Z 187,A 147.0819,B 2.4279,C 0.0679,E1 2.2986,E2 306.7643} C_DIS
LIN {X -113.4689,Y 80.7553,Z 187,A 145.6031,B 2.4281,C 0.0628,E1 2.3009,E2 308.1978} C_DIS
LIN {X -110.9036,Y 84.2443,Z 187,A 143.68,B 2.4281,C 0.0593,E1 2.3042,E2 310.1371} C_DIS
LIN {X -107.955,Y 87.9902,Z 187,A 141.6824,B 2.4283,C 0.0552,E1 2.3077,E2 312.1377} C_DIS
LIN {X -105.2378,Y 91.2234,Z 187,A 139.5394,B 2.4283,C 0.0528,E1 2.3117,E2 314.3291} C_DIS
LIN {X -102.7134,Y 94.0561,Z 187,A 138.491,B 2.4284,C 0.0482,E1 2.3135,E2 315.3135} C_DIS
LIN {X -100.4832,Y 96.4351,Z 187,A 136.8292,B 2.4284,C 0.0465,E1 2.3168,E2 317.0138} C_DIS
LIN {X -97.4171,Y 99.5311,Z 187,A 134.9543,B 2.4285,C 0.0433,E1 2.3205,E2 318.8974} C_DIS
LIN {X -92.4721,Y 104.1418,Z 187,A 132.038,B 2.4285,C 0.0387,E1 2.3266,E2 321.8282} C_DIS
LIN {X -89.0988,Y 107.0422,Z 187,A 130.1074,B 2.4286,C 0.0359,E1 2.3307,E2 323.7698} C_DIS
LIN {X -85.6879,Y 109.792,Z 187,A 127.6623,B 2.4286,C 0.0351,E1 2.3363,E2 326.2914} C_DIS
LIN {X -81.2709,Y 113.1003,Z 187,A 126.1653,B 2.4287,C 0.029,E1 2.3394,E2 327.6932} C_DIS
LIN {X -78.4633,Y 115.0661,Z 187,A 124.4814,B 2.4287,C 0.0278,E1 2.3434,E2 329.4095} C_DIS
LIN {X -75.775,Y 116.8532,Z 187,A 123.1581,B 2.4287,C 0.0259,E1 2.3465,E2 330.7314} C_DIS
LIN {X -72.2868,Y 119.0429,Z 187,A 121.1536,B 2.4287,C 0.0248,E1 2.3513,E2 332.7723} C_DIS
LIN {X -69.3424,Y 120.782,Z 187,A 120.0338,B 2.4287,C 0.0219,E1 2.3539,E2 333.8564} C_DIS
LIN {X -65.8839,Y 122.7022,Z 187,A 118.1675,B 2.4287,C 0.0208,E1 2.3586,E2 335.7506} C_DIS
LIN {X -60.9513,Y 125.2255,Z 187,A 115.9931,B 2.4288,C 0.0179,E1 2.364,E2 337.9108} C_DIS
LIN {X -56.8847,Y 127.1224,Z 187,A 114.0193,B 2.4288,C 0.0165,E1 2.3691,E2 339.8989} C_DIS
LIN {X -52.7872,Y 128.8801,Z 187,A 112.2911,B 2.4288,C 0.0143,E1 2.3735,E2 341.6131} C_DIS
LIN {X -48.6081,Y 130.5117,Z 187,A 110.2385,B 2.4288,C 0.0136,E1 2.3789,E2 343.6896} C_DIS
LIN {X -43.6545,Y 132.2513,Z 187,A 108.1792,B 2.4288,C 0.0115,E1 2.3843,E2 345.7355} C_DIS
LIN {X -39.7309,Y 133.4835,Z 187,A 106.5567,B 2.4288,C 0.01,E1 2.3886,E2 347.3487} C_DIS
LIN {X -36.5324,Y 134.3944,Z 187,A 105.153,B 2.4288,C 0.0094,E1 2.3924,E2 348.7559} C_DIS
LIN {X -34.0241,Y 135.0498,Z 187,A 104.0162,B 2.4288,C 0.0091,E1 2.3955,E2 349.9006} C_DIS
LIN {X -29.9942,Y 136.0028,Z 187,A 102.3729,B 2.4288,C 0.008,E1 2.4,E2 351.5357} C_DIS
LIN {X -26.9105,Y 136.6472,Z 187,A 101.0077,B 2.4288,C 0.0078,E1 2.4037,E2 352.9087} C_DIS
LIN {X -23.8999,Y 137.2052,Z 187,A 99.6923,B 2.4288,C 0.0077,E1 2.4074,E2 354.2302} C_DIS
LIN {X -18.8569,Y 137.9894,Z 187,A 97.631,B 2.4288,C 0.007,E1 2.4131,E2 356.2858} C_DIS
LIN {X -15.3318,Y 138.424,Z 187,A 95.7542,B 2.4288,C 0.0088,E1 2.4184,E2 358.2119} C_DIS
LIN {X -11.6322,Y 138.7832,Z 187,A 94.1844,B 2.4288,C 0.0089,E1 2.4228,E2 359.7857} C_DIS
LIN {X -7.5835,Y 139.0645,Z 187,A 93.0267,B 2.4288,C 0.0063,E1 2.4259,E2 360.8812} C_DIS
LIN {X -4.5461,Y 139.1974,Z 187,A 91.5727,B 2.4288,C 0.0074,E1 2.43,E2 362.3592} C_DIS
LIN {X -0.6753,Y 139.2684,Z 187,A 90.0556,B 2.4288,C 0.0072,E1 2.4342,E2 363.8664} C_DIS
LIN {X 2.6243,Y 139.2456,Z 187,A 88.7692,B 2.4288,C 0.0072,E1 2.4378,E2 365.1437} C_DIS
LIN {X 6.3157,Y 139.1283,Z 187,A 87.1329,B 2.4288,C 0.0082,E1 2.4424,E2 366.7936} C_DIS
LIN {X 10.0415,Y 138.9074,Z 187,A 85.7009,B 2.4288,C 0.0082,E1 2.4464,E2 368.2125} C_DIS
LIN {X 13.6185,Y 138.6027,Z 187,A 84.1931,B 2.4288,C 0.0089,E1 2.4506,E2 369.7235} C_DIS
LIN {X 17.9426,Y 138.1092,Z 187,A 81.7519,B 2.4288,C 0.0136,E1 2.4576,E2 372.2422} C_DIS
LIN {X 23.6305,Y 137.2522,Z 187,A 79.0355,B 2.4288,C 0.0171,E1 2.4652,E2 374.9995} C_DIS
LIN {X 31.1888,Y 135.7325,Z 187,A 76.9785,B 2.4288,C 0.0129,E1 2.4704,E2 376.922} C_DIS
LIN {X 34.1524,Y 135.0172,Z 187,A 75.7609,B 2.4288,C 0.0137,E1 2.4737,E2 378.1349} C_DIS
LIN {X 37.4793,Y 134.1317,Z 187,A 74.3756,B 2.4288,C 0.0148,E1 2.4775,E2 379.5161} C_DIS
LIN {X 41.559,Y 132.9267,Z 187,A 72.6784,B 2.4288,C 0.0161,E1 2.482,E2 381.2065} C_DIS
LIN {X 45.2435,Y 131.7163,Z 187,A 71.2707,B 2.4288,C 0.0166,E1 2.4857,E2 382.591} C_DIS
LIN {X 49.1205,Y 130.3198,Z 187,A 69.3648,B 2.4288,C 0.0198,E1 2.4907,E2 384.5222} C_DIS
LIN {X 52.9473,Y 128.8145,Z 187,A 67.5865,B 2.4288,C 0.0224,E1 2.4954,E2 386.3109} C_DIS
LIN {X 56.9187,Y 127.1071,Z 187,A 66.0242,B 2.4288,C 0.0232,E1 2.4993,E2 387.8465} C_DIS
LIN {X 63.146,Y 124.1311,Z 187,A 63.5231,B 2.4288,C 0.0248,E1 2.5055,E2 390.3059} C_DIS
LIN {X 65.8616,Y 122.7142,Z 187,A 61.9865,B 2.4288,C 0.0285,E1 2.5094,E2 391.8764} C_DIS
LIN {X 69.8499,Y 120.4887,Z 187,A 60.2066,B 2.4287,C 0.0307,E1 2.5137,E2 393.644} C_DIS
LIN {X 73.2764,Y 118.4366,Z 187,A 58.5905,B 2.4287,C 0.0331,E1 2.5175,E2 395.2567} C_DIS
LIN {X 77.0464,Y 116.0189,Z 187,A 56.4651,B 2.4286,C 0.0381,E1 2.5226,E2 397.4167} C_DIS
LIN {X 80.4469,Y 113.6875,Z 187,A 55.417,B 2.4286,C 0.0364,E1 2.5248,E2 398.3853} C_DIS
LIN {X 82.7522,Y 112.0211,Z 187,A 54.0238,B 2.4286,C 0.0401,E1 2.528,E2 399.806} C_DIS
LIN {X 86.4202,Y 109.2164,Z 187,A 52.1736,B 2.4286,C 0.0432,E1 2.5321,E2 401.6502} C_DIS
LIN {X 90.496,Y 105.8638,Z 187,A 50.2103,B 2.4285,C 0.0458,E1 2.5362,E2 403.588} C_DIS
LIN {X 96.3259,Y 100.5875,Z 187,A 47.2805,B 2.4284,C 0.0499,E1 2.5422,E2 406.4804} C_DIS
LIN {X 99.7858,Y 97.1569,Z 187,A 45.0729,B 2.4283,C 0.0556,E1 2.5466,E2 408.7135} C_DIS
LIN {X 102.9117,Y 93.8393,Z 187,A 43.1345,B 2.4281,C 0.0601,E1 2.5503,E2 410.66} C_DIS
LIN {X 105.9498,Y 90.3948,Z 187,A 40.7476,B 2.4279,C 0.0681,E1 2.5548,E2 413.1086} C_DIS
LIN {X 110.0235,Y 85.3894,Z 187,A 39.2392,B 2.428,C 0.0652,E1 2.5571,E2 414.4755} C_DIS
LIN {X 112.967,Y 81.456,Z 187,A 37.0229,B 2.4278,C 0.0714,E1 2.5609,E2 416.7166} C_DIS
LIN {X 115.5293,Y 77.7794,Z 187,A 35.2611,B 2.4278,C 0.0751,E1 2.5636,E2 418.4687} C_DIS
LIN {X 118.0116,Y 73.9593,Z 187,A 33.4418,B 2.4276,C 0.0792,E1 2.5664,E2 420.2816} C_DIS
LIN {X 120.4016,Y 70.0003,Z 187,A 31.6863,B 2.4275,C 0.0826,E1 2.5688,E2 422.0193} C_DIS
LIN {X 122.4952,Y 66.2693,Z 187,A 29.9767,B 2.4273,C 0.0866,E1 2.5711,E2 423.7231} C_DIS
LIN {X 124.3345,Y 62.7464,Z 187,A 28.4296,B 2.4273,C 0.09,E1 2.5731,E2 425.2597} C_DIS
LIN {X 125.9571,Y 59.424,Z 187,A 27.095,B 2.4271,C 0.0924,E1 2.5747,E2 426.5712} C_DIS
LIN {X 127.3773,Y 56.3148,Z 187,A 25.6183,B 2.427,C 0.0966,E1 2.5764,E2 428.0573} C_DIS
LIN {X 129.0771,Y 52.2984,Z 187,A 23.9706,B 2.4268,C 0.1001,E1 2.5781,E2 429.6871} C_DIS
LIN {X 130.7262,Y 48.0352,Z 187,A 22.2712,B 2.4267,C 0.1036,E1 2.5798,E2 431.3645} C_DIS
LIN {X 131.6752,Y 45.362,Z 187,A 21.1608,B 2.4266,C 0.1062,E1 2.5808,E2 432.4681} C_DIS
LIN {X 132.7229,Y 42.1979,Z 187,A 19.813,B 2.4264,C 0.1097,E1 2.5819,E2 433.8134} C_DIS
LIN {X 134.03,Y 37.8428,Z 187,A 18.0007,B 2.4262,C 0.1143,E1 2.5834,E2 435.6193} C_DIS
LIN {X 134.9654,Y 34.3566,Z 187,A 16.6786,B 2.4261,C 0.117,E1 2.5843,E2 436.9213} C_DIS
LIN {X 135.8531,Y 30.661,Z 187,A 15.1968,B 2.4259,C 0.1206,E1 2.5852,E2 438.3933} C_DIS
LIN {X 136.6901,Y 26.6861,Z 187,A 12.9578,B 2.4254,C 0.13,E1 2.5865,E2 440.7057} C_DIS
LIN {X 137.6489,Y 21.186,Z 187,A 11.4753,B 2.4254,C 0.1295,E1 2.5871,E2 442.0853} C_DIS
LIN {X 138.0961,Y 18.0424,Z 187,A 10.2103,B 2.4253,C 0.1327,E1 2.5875,E2 443.3458} C_DIS
LIN {X 138.563,Y 14.0325,Z 187,A 8.6971,B 2.4251,C 0.1361,E1 2.588,E2 444.8409} C_DIS
LIN {X 138.9512,Y 9.4417,Z 187,A 6.7474,B 2.4247,C 0.1419,E1 2.5884,E2 446.7986} C_DIS
LIN {X 139.165,Y 5.4061,Z 187,A 5.2998,B 2.4246,C 0.1447,E1 2.5886,E2 448.2193} C_DIS
LIN {X 139.263,Y 1.5764,Z 187,A 3.8228,B 2.4244,C 0.1483,E1 2.5886,E2 449.6845} C_DIS
LIN {X 139.2547,Y -2.0741,Z 187,A 2.411,B 2.4241,C 0.1517,E1 2.5886,E2 451.0855} C_DIS
LIN {X 139.1635,Y -5.4443,Z 187,A 1.0464,B 2.4239,C 0.1554,E1 2.5886,E2 452.4481} C_DIS
LIN {X 138.9284,Y -9.7548,Z 187,A -0.6445,B 2.4236,C 0.1597,E1 2.5883,E2 454.1291} C_DIS
LIN {X 138.6259,Y -13.3774,Z 187,A -2.0269,B 2.4234,C 0.1629,E1 2.5879,E2 455.4977} C_DIS
LIN {X 138.1857,Y -17.3588,Z 187,A -3.5382,B 2.4232,C 0.1663,E1 2.5874,E2 456.9923} C_DIS
LIN {X 137.8397,Y -19.9081,Z 187,A -4.7509,B 2.4229,C 0.1706,E1 2.5869,E2 458.2258} C_DIS
LIN {X 137.2845,Y -23.4373,Z 187,A -6.1417,B 2.4226,C 0.174,E1 2.5863,E2 459.6074} C_DIS
LIN {X 135.8789,Y -30.5479,Z 187,A -8.6566,B 2.4223,C 0.1782,E1 2.585,E2 462.063} C_DIS
LIN {X 134.578,Y -35.8439,Z 187,A -10.6409,B 2.4221,C 0.1822,E1 2.5836,E2 464.0146} C_DIS
LIN {X 134.0788,Y -37.6685,Z 187,A -11.6555,B 2.4217,C 0.1863,E1 2.5829,E2 465.0611} C_DIS
LIN {X 132.8744,Y -41.7237,Z 187,A -13.2364,B 2.4215,C 0.1897,E1 2.5816,E2 466.6223} C_DIS
LIN {X 132.0005,Y -44.4077,Z 187,A -14.4284,B 2.4212,C 0.193,E1 2.5805,E2 467.8192} C_DIS
LIN {X 130.6461,Y -48.2494,Z 187,A -15.9079,B 2.421,C 0.1958,E1 2.5792,E2 469.2739} C_DIS
LIN {X 129.6979,Y -50.7397,Z 187,A -17.039,B 2.4207,C 0.199,E1 2.578,E2 470.4104} C_DIS
LIN {X 128.0678,Y -54.7262,Z 187,A -18.6824,B 2.4204,C 0.2026,E1 2.5763,E2 472.0382} C_DIS
LIN {X 126.2722,Y -58.7485,Z 187,A -20.3801,B 2.4201,C 0.2063,E1 2.5743,E2 473.722} C_DIS
LIN {X 124.9246,Y -61.5613,Z 187,A -21.7662,B 2.4198,C 0.2105,E1 2.5726,E2 475.1228} C_DIS
LIN {X 123.1223,Y -65.0921,Z 187,A -23.2157,B 2.4195,C 0.2131,E1 2.5708,E2 476.5494} C_DIS
LIN {X 120.189,Y -70.3645,Z 187,A -25.6515,B 2.419,C 0.2189,E1 2.5674,E2 478.9809} C_DIS
LIN {X 117.7711,Y -74.3404,Z 187,A -27.4681,B 2.4187,C 0.2228,E1 2.5648,E2 480.7859} C_DIS
LIN {X 114.984,Y -78.5829,Z 187,A -29.4578,B 2.4183,C 0.2269,E1 2.5617,E2 482.7641} C_DIS
LIN {X 111.3154,Y -83.6986,Z 187,A -31.9366,B 2.4178,C 0.2321,E1 2.5577,E2 485.2301} C_DIS
LIN {X 108.5461,Y -87.26,Z 187,A -33.6129,B 2.4175,C 0.2348,E1 2.5548,E2 486.8837} C_DIS
LIN {X 105.8588,Y -90.5018,Z 187,A -35.4233,B 2.4171,C 0.2393,E1 2.5515,E2 488.706} C_DIS
LIN {X 102.8387,Y -93.9197,Z 187,A -37.1351,B 2.4168,C 0.2421,E1 2.5483,E2 490.3971} C_DIS
LIN {X 99.747,Y -97.1969,Z 187,A -38.8627,B 2.4165,C 0.245,E1 2.545,E2 492.1092} C_DIS
LIN {X 96.6786,Y -100.2488,Z 187,A -40.71,B 2.4161,C 0.2492,E1 2.5413,E2 493.9669} C_DIS
LIN {X 92.8677,Y -103.7888,Z 187,A -42.6108,B 2.4158,C 0.2516,E1 2.5375,E2 495.8369} C_DIS
LIN {X 89.7462,Y -106.4999,Z 187,A -44.3313,B 2.4155,C 0.2551,E1 2.5338,E2 497.5614} C_DIS
LIN {X 86.2498,Y -109.3507,Z 187,A -46.1983,B 2.4151,C 0.2586,E1 2.5297,E2 499.4314} C_DIS
LIN {X 81.9644,Y -112.5986,Z 187,A -48.2626,B 2.4148,C 0.2615,E1 2.5251,E2 501.4774} C_DIS
LIN {X 78.1374,Y -115.2869,Z 187,A -50.0458,B 2.4145,C 0.2637,E1 2.5211,E2 503.2428} C_DIS
LIN {X 74.8571,Y -117.4436,Z 187,A -51.792,B 2.4141,C 0.2674,E1 2.5169,E2 505.008} C_DIS
LIN {X 70.2093,Y -120.2802,Z 187,A -53.8411,B 2.4139,C 0.2695,E1 2.5121,E2 507.0329} C_DIS
LIN {X 66.2756,Y -122.4918,Z 187,A -55.671,B 2.4136,C 0.2721,E1 2.5076,E2 508.8606} C_DIS
LIN {X 62.972,Y -124.2197,Z 187,A -57.0715,B 2.4135,C 0.2733,E1 2.5041,E2 510.2439} C_DIS
LIN {X 59.8807,Y -125.739,Z 187,A -58.4627,B 2.4133,C 0.2751,E1 2.5007,E2 511.6325} C_DIS
LIN {X 56.6486,Y -127.228,Z 187,A -59.8367,B 2.4131,C 0.2764,E1 2.4972,E2 512.9953} C_DIS
LIN {X 53.2621,Y -128.683,Z 187,A -61.3141,B 2.4129,C 0.278,E1 2.4934,E2 514.4684} C_DIS
LIN {X 48.4107,Y -130.5856,Z 187,A -63.3511,B 2.4127,C 0.2798,E1 2.4881,E2 516.4923} C_DIS
LIN {X 45.5275,Y -131.6178,Z 187,A -64.633,B 2.4125,C 0.2813,E1 2.4847,E2 517.778} C_DIS
LIN {X 42.2237,Y -132.7147,Z 187,A -66.036,B 2.4124,C 0.2826,E1 2.481,E2 519.1779} C_DIS
LIN {X 38.8871,Y -133.7306,Z 187,A -67.4251,B 2.4123,C 0.2837,E1 2.4773,E2 520.5617} C_DIS
LIN {X 35.0604,Y -134.7868,Z 187,A -69.4923,B 2.4117,C 0.2882,E1 2.4715,E2 522.6893} C_DIS
LIN {X 31.0221,Y -135.7706,Z 187,A -70.4099,B 2.4122,C 0.2843,E1 2.4693,E2 523.4995} C_DIS
LIN {X 23.8413,Y -137.2157,Z 187,A -73.6944,B 2.4117,C 0.2883,E1 2.4602,E2 526.8231} C_DIS
LIN {X 17.3588,Y -138.1857,Z 187,A -76.3061,B 2.4117,C 0.2894,E1 2.453,E2 529.4247} C_DIS
LIN {X 13.1961,Y -138.6433,Z 187,A -78.0717,B 2.4115,C 0.2905,E1 2.4481,E2 531.1971} C_DIS
LIN {X 9.7384,Y -138.9296,Z 187,A -79.4014,B 2.4115,C 0.2905,E1 2.4444,E2 532.5142} C_DIS
LIN {X 6.9045,Y -139.0987,Z 187,A -80.6647,B 2.4113,C 0.2915,E1 2.4408,E2 533.7912} C_DIS
LIN {X 3.5087,Y -139.2262,Z 187,A -81.9772,B 2.4113,C 0.2913,E1 2.4372,E2 535.0927} C_DIS
LIN {X 0.9877,Y -139.2619,Z 187,A -82.7915,B 2.4115,C 0.2902,E1 2.435,E2 535.8767} C_DIS
Enddeposition()
LIN {X 0.9877,Y -139.2619,Z 187,A -82.7915,B 2.4115,C 0.2902,E1 2.435,E2 535.8767} C_DIS
Startdeposition()
$VEL.CP = VEL_PRINT
LIN {X 1.7724,Y -140.1596,Z 187,A -82.0115,B 2.4154,C 0.2888,E1 2.441,E2 535.0615} C_DIS
LIN {X 5.8053,Y -140.0498,Z 187,A -80.3969,B 2.4154,C 0.2885,E1 2.4455,E2 533.4509} C_DIS
LIN {X 10.0511,Y -139.8088,Z 187,A -78.6824,B 2.4155,C 0.288,E1 2.4503,E2 531.7387} C_DIS
LIN {X 13.9611,Y -139.4737,Z 187,A -77.0856,B 2.4156,C 0.2873,E1 2.4547,E2 530.1422} C_DIS
LIN {X 17.5332,Y -139.0702,Z 187,A -75.7294,B 2.4156,C 0.2873,E1 2.4585,E2 528.801} C_DIS
LIN {X 21.5157,Y -138.5083,Z 187,A -73.9509,B 2.4158,C 0.2854,E1 2.4634,E2 527.0027} C_DIS
LIN {X 28.0256,Y -137.3391,Z 187,A -71.4071,B 2.4159,C 0.2845,E1 2.4704,E2 524.4796} C_DIS
LIN {X 31.238,Y -136.6442,Z 187,A -70.1143,B 2.416,C 0.2838,E1 2.4739,E2 523.1931} C_DIS
LIN {X 35.0338,Y -135.7217,Z 187,A -68.4378,B 2.4163,C 0.2819,E1 2.4785,E2 521.5045} C_DIS
LIN {X 39.0245,Y -134.6278,Z 187,A -66.8571,B 2.4163,C 0.281,E1 2.4827,E2 519.9382} C_DIS
LIN {X 42.6588,Y -133.5201,Z 187,A -65.3418,B 2.4165,C 0.2797,E1 2.4867,E2 518.4271} C_DIS
LIN {X 45.9126,Y -132.4365,Z 187,A -63.9634,B 2.4167,C 0.2784,E1 2.4904,E2 517.051} C_DIS
LIN {X 50.9915,Y -130.5653,Z 187,A -61.7654,B 2.4169,C 0.2759,E1 2.4961,E2 514.8536} C_DIS
LIN {X 54.9395,Y -128.9558,Z 187,A -60.1359,B 2.4171,C 0.2746,E1 2.5003,E2 513.2387} C_DIS
LIN {X 59.1314,Y -127.0864,Z 187,A -58.2448,B 2.4174,C 0.272,E1 2.5051,E2 511.3442} C_DIS
LIN {X 62.7382,Y -125.3472,Z 187,A -56.4983,B 2.4177,C 0.2689,E1 2.5096,E2 509.5812} C_DIS
LIN {X 66.6587,Y -123.3072,Z 187,A -54.8371,B 2.4179,C 0.2673,E1 2.5136,E2 507.939} C_DIS
LIN {X 70.5222,Y -121.139,Z 187,A -53.1653,B 2.4181,C 0.2656,E1 2.5176,E2 506.2852} C_DIS
LIN {X 76.8951,Y -117.1969,Z 187,A -50.1305,B 2.4186,C 0.2608,E1 2.5248,E2 503.2522} C_DIS
LIN {X 80.5564,Y -114.7113,Z 187,A -48.4545,B 2.4188,C 0.2587,E1 2.5286,E2 501.5932} C_DIS
LIN {X 85.0989,Y -111.3827,Z 187,A -45.5887,B 2.4198,C 0.2501,E1 2.5352,E2 498.6473} C_DIS
LIN {X 89.421,Y -107.9436,Z 187,A -44.0009,B 2.4196,C 0.2511,E1 2.5384,E2 497.1509} C_DIS
LIN {X 92.4285,Y -105.3804,Z 187,A -41.9703,B 2.4203,C 0.2446,E1 2.5428,E2 495.0615} C_DIS
LIN {X 96.0466,Y -102.0931,Z 187,A -40.1364,B 2.4206,C 0.2419,E1 2.5465,E2 493.2489} C_DIS
LIN {X 99.2247,Y -99.0074,Z 187,A -38.7795,B 2.4206,C 0.2419,E1 2.5491,E2 491.9533} C_DIS
LIN {X 102.3293,Y -95.7955,Z 187,A -37.0618,B 2.4209,C 0.2388,E1 2.5524,E2 490.2491} C_DIS
LIN {X 107.2629,Y -90.2365,Z 187,A -34.1015,B 2.4215,C 0.2328,E1 2.5578,E2 487.2972} C_DIS
LIN {X 110.1017,Y -86.7501,Z 187,A -32.3611,B 2.4218,C 0.2294,E1 2.5608,E2 485.5687} C_DIS
LIN {X 111.9123,Y -84.4012,Z 187,A -31.0764,B 2.4221,C 0.226,E1 2.563,E2 484.2731} C_DIS
LIN {X 115.2958,Y -79.7181,Z 187,A -29.0506,B 2.4224,C 0.2233,E1 2.5662,E2 482.2915} C_DIS
LIN {X 117.5912,Y -76.2905,Z 187,A -27.3496,B 2.4228,C 0.2191,E1 2.5688,E2 480.5871} C_DIS
LIN {X 120.0778,Y -72.3141,Z 187,A -25.533,B 2.4231,C 0.2153,E1 2.5715,E2 478.7827} C_DIS
LIN {X 122.1961,Y -68.6735,Z 187,A -23.352,B 2.4238,C 0.207,E1 2.5746,E2 476.5375} C_DIS
LIN {X 124.7099,Y -63.9923,Z 187,A -21.9266,B 2.4238,C 0.2079,E1 2.5763,E2 475.2124} C_DIS
LIN {X 126.4881,Y -60.3997,Z 187,A -19.9403,B 2.4243,C 0.2007,E1 2.5787,E2 473.1775} C_DIS
LIN {X 128.2921,Y -56.473,Z 187,A -18.5487,B 2.4245,C 0.1994,E1 2.5802,E2 471.8357} C_DIS
LIN {X 129.8975,Y -52.6697,Z 187,A -17.0719,B 2.4247,C 0.1968,E1 2.5818,E2 470.386} C_DIS
LIN {X 131.4135,Y -48.7653,Z 187,A -15.1046,B 2.4252,C 0.19,E1 2.5838,E2 468.3829} C_DIS
LIN {X 132.7268,Y -45.0742,Z 187,A -13.8841,B 2.4252,C 0.189,E1 2.5848,E2 467.2129} C_DIS
LIN {X 133.9588,Y -41.2614,Z 187,A -12.2958,B 2.4256,C 0.185,E1 2.5861,E2 465.6299} C_DIS
LIN {X 135.2429,Y -36.8414,Z 187,A -9.8718,B 2.4263,C 0.1751,E1 2.588,E2 463.1312} C_DIS
LIN {X 136.6877,Y -31.0473,Z 187,A -7.649,B 2.4267,C 0.1703,E1 2.5893,E2 460.9362} C_DIS
LIN {X 137.8296,Y -25.5164,Z 187,A -5.9758,B 2.4267,C 0.1696,E1 2.5902,E2 459.3471} C_DIS
LIN {X 138.4679,Y -21.7766,Z 187,A -4.7037,B 2.4268,C 0.1677,E1 2.5907,E2 458.1113} C_DIS
LIN {X 138.945,Y -18.489,Z 187,A -3.3201,B 2.4271,C 0.1637,E1 2.5913,E2 456.7233} C_DIS
LIN {X 139.396,Y -14.7077,Z 187,A -1.8405,B 2.4274,C 0.16,E1 2.5917,E2 455.2528} C_DIS
LIN {X 139.7698,Y -10.5856,Z 187,A -0.3109,B 2.4276,C 0.1567,E1 2.5921,E2 453.7438} C_DIS
LIN {X 139.9909,Y -7.0757,Z 187,A 0.9843,B 2.4278,C 0.1539,E1 2.5923,E2 452.4665} C_DIS
LIN {X 140.1453,Y -2.6297,Z 187,A 2.8123,B 2.4281,C 0.1487,E1 2.5924,E2 450.6362} C_DIS
LIN {X 140.1663,Y 0.9965,Z 187,A 4.223,B 2.4283,C 0.1451,E1 2.5924,E2 449.234} C_DIS
LIN {X 140.0651,Y 5.4108,Z 187,A 5.9047,B 2.4285,C 0.1411,E1 2.5923,E2 447.5675} C_DIS
LIN {X 139.8612,Y 9.3198,Z 187,A 7.4482,B 2.4288,C 0.1371,E1 2.592,E2 446.0305} C_DIS
LIN {X 139.5354,Y 13.318,Z 187,A 8.9925,B 2.429,C 0.1334,E1 2.5917,E2 444.4978} C_DIS
LIN {X 139.0778,Y 17.4752,Z 187,A 10.5924,B 2.4292,C 0.1296,E1 2.5911,E2 442.9114} C_DIS
LIN {X 138.4333,Y 21.9998,Z 187,A 12.4277,B 2.4294,C 0.1246,E1 2.5904,E2 441.0794} C_DIS
LIN {X 137.3367,Y 28.0373,Z 187,A 15.0148,B 2.4298,C 0.117,E1 2.589,E2 438.4806} C_DIS
LIN {X 136.5868,Y 31.4889,Z 187,A 16.1168,B 2.4298,C 0.116,E1 2.5884,E2 437.4227} C_DIS
LIN {X 135.7371,Y 34.9731,Z 187,A 17.9226,B 2.4302,C 0.1091,E1 2.5871,E2 435.5717} C_DIS
LIN {X 134.5805,Y 39.1861,Z 187,A 19.0431,B 2.4302,C 0.11,E1 2.5863,E2 434.5373} C_DIS
LIN {X 133.5481,Y 42.5714,Z 187,A 20.5126,B 2.4303,C 0.1058,E1 2.5851,E2 433.0642} C_DIS
LIN {X 132.4919,Y 45.7527,Z 187,A 21.822,B 2.4305,C 0.1027,E1 2.5839,E2 431.7621} C_DIS
LIN {X 131.4558,Y 48.6525,Z 187,A 23.0937,B 2.4306,C 0.0992,E1 2.5827,E2 430.4883} C_DIS
LIN {X 130.1674,Y 52.0003,Z 187,A 24.4264,B 2.4307,C 0.0965,E1 2.5813,E2 429.1722} C_DIS
LIN {X 128.908,Y 55.0499,Z 187,A 25.7393,B 2.4308,C 0.0933,E1 2.5799,E2 427.8634} C_DIS
LIN {X 127.3803,Y 58.4959,Z 187,A 27.1549,B 2.431,C 0.0903,E1 2.5783,E2 426.4634} C_DIS
LIN {X 125.8449,Y 61.7293,Z 187,A 28.5938,B 2.431,C 0.0868,E1 2.5765,E2 425.0271} C_DIS
LIN {X 124.1411,Y 65.0872,Z 187,A 29.9523,B 2.4312,C 0.0844,E1 2.5748,E2 423.6913} C_DIS
LIN {X 122.1427,Y 68.7685,Z 187,A 31.7151,B 2.4313,C 0.0797,E1 2.5724,E2 421.9215} C_DIS
LIN {X 119.7776,Y 72.8104,Z 187,A 33.533,B 2.4315,C 0.0758,E1 2.5699,E2 420.1155} C_DIS
LIN {X 117.3761,Y 76.6218,Z 187,A 35.3155,B 2.4315,C 0.0719,E1 2.5672,E2 418.34} C_DIS
LIN {X 114.828,Y 80.3904,Z 187,A 37.089,B 2.4317,C 0.0682,E1 2.5644,E2 416.577} C_DIS
LIN {X 112.1233,Y 84.1216,Z 187,A 38.8189,B 2.4317,C 0.065,E1 2.5615,E2 414.8664} C_DIS
LIN {X 109.7326,Y 87.2157,Z 187,A 40.6026,B 2.4319,C 0.0599,E1 2.5584,E2 413.0585} C_DIS
LIN {X 107.5045,Y 89.9485,Z 187,A 41.779,B 2.4319,C 0.0588,E1 2.5564,E2 411.9157} C_DIS
LIN {X 105.1466,Y 92.6939,Z 187,A 43.1798,B 2.4319,C 0.0562,E1 2.5538,E2 410.5247} C_DIS
LIN {X 102.1999,Y 95.9335,Z 187,A 44.9212,B 2.4321,C 0.0528,E1 2.5505,E2 408.7893} C_DIS
LIN {X 98.9954,Y 99.2367,Z 187,A 46.7261,B 2.4321,C 0.0494,E1 2.547,E2 406.9937} C_DIS
LIN {X 96.7148,Y 101.4604,Z 187,A 48.0265,B 2.4321,C 0.0468,E1 2.5444,E2 405.6934} C_DIS
LIN {X 92.1046,Y 105.663,Z 187,A 50.3624,B 2.4322,C 0.0434,E1 2.5396,E2 403.3844} C_DIS
LIN {X 88.6839,Y 108.5499,Z 187,A 52.1597,B 2.4322,C 0.0402,E1 2.5357,E2 401.5911} C_DIS
LIN {X 85.0141,Y 111.4476,Z 187,A 53.9828,B 2.4323,C 0.0374,E1 2.5317,E2 399.7791} C_DIS
LIN {X 81.4976,Y 114.0442,Z 187,A 55.5335,B 2.4323,C 0.036,E1 2.5283,E2 398.2579} C_DIS
LIN {X 77.8991,Y 116.5319,Z 187,A 57.4518,B 2.4324,C 0.032,E1 2.5238,E2 396.3234} C_DIS
LIN {X 74.0908,Y 118.9894,Z 187,A 59.2213,B 2.4324,C 0.0296,E1 2.5196,E2 394.5644} C_DIS
LIN {X 70.3005,Y 121.2674,Z 187,A 60.9971,B 2.4324,C 0.027,E1 2.5154,E2 392.7926} C_DIS
LIN {X 66.1717,Y 123.5689,Z 187,A 62.856,B 2.4325,C 0.0247,E1 2.5108,E2 390.9431} C_DIS
LIN {X 62.9502,Y 125.2403,Z 187,A 64.5504,B 2.4325,C 0.0212,E1 2.5065,E2 389.2224} C_DIS
LIN {X 59.6486,Y 126.847,Z 187,A 65.8125,B 2.4325,C 0.0208,E1 2.5034,E2 387.9905} C_DIS
LIN {X 55.9173,Y 128.533,Z 187,A 67.1469,B 2.4325,C 0.0209,E1 2.5001,E2 386.6985} C_DIS
LIN {X 52.738,Y 129.87,Z 187,A 68.5695,B 2.4325,C 0.0191,E1 2.4964,E2 385.2745} C_DIS
LIN {X 49.3468,Y 131.1957,Z 187,A 70.1914,B 2.4325,C 0.0166,E1 2.4922,E2 383.6362} C_DIS
LIN {X 45.9658,Y 132.418,Z 187,A 72.198,B 2.4326,C 0.0115,E1 2.4867,E2 381.5628} C_DIS
LIN {X 40.9863,Y 134.043,Z 187,A 73.6495,B 2.4326,C 0.0138,E1 2.483,E2 380.1979} C_DIS
LIN {X 37.7619,Y 134.9869,Z 187,A 75.0241,B 2.4326,C 0.0125,E1 2.4793,E2 378.8235} C_DIS
LIN {X 34.5803,Y 135.8368,Z 187,A 76.7256,B 2.4326,C 0.0092,E1 2.4746,E2 377.0782} C_DIS
LIN {X 30.7588,Y 136.7536,Z 187,A 77.9208,B 2.4326,C 0.0105,E1 2.4715,E2 375.9345} C_DIS
LIN {X 26.6823,Y 137.6068,Z 187,A 79.631,B 2.4326,C 0.0092,E1 2.4668,E2 374.2239} C_DIS
LIN {X 23.2423,Y 138.2291,Z 187,A 81.1738,B 2.4326,C 0.0076,E1 2.4625,E2 372.6674} C_DIS
LIN {X 18.3977,Y 138.9569,Z 187,A 83.0133,B 2.4326,C 0.0074,E1 2.4575,E2 370.8488} C_DIS
LIN {X 14.5241,Y 139.4158,Z 187,A 84.6566,B 2.4326,C 0.0064,E1 2.4529,E2 369.2001} C_DIS
LIN {X 10.4532,Y 139.7795,Z 187,A 86.1852,B 2.4326,C 0.0066,E1 2.4487,E2 367.6896} C_DIS
LIN {X 7.1165,Y 139.9888,Z 187,A 87.6025,B 2.4326,C 0.0058,E1 2.4447,E2 366.2665} C_DIS
LIN {X 3.458,Y 140.1276,Z 187,A 89.0735,B 2.4326,C 0.0056,E1 2.4406,E2 364.7993} C_DIS
LIN {X -0.4447,Y 140.1694,Z 187,A 90.6986,B 2.4326,C 0.0051,E1 2.436,E2 363.1711} C_DIS
LIN {X -4.1575,Y 140.1082,Z 187,A 92.2728,B 2.4326,C 0.0047,E1 2.4316,E2 361.5906} C_DIS
LIN {X -7.4406,Y 139.9725,Z 187,A 93.6207,B 2.4326,C 0.0047,E1 2.4278,E2 360.2428} C_DIS
LIN {X -12.9318,Y 139.5725,Z 187,A 95.8863,B 2.4326,C 0.0047,E1 2.4215,E2 357.9764} C_DIS
LIN {X -17.1125,Y 139.1219,Z 187,A 97.5657,B 2.4326,C 0.0052,E1 2.4169,E2 356.3027} C_DIS
LIN {X -25.3702,Y 137.856,Z 187,A 101.1236,B 2.4326,C 0.0055,E1 2.407,E2 352.729} C_DIS
LIN {X -29.9749,Y 136.9274,Z 187,A 102.9183,B 2.4326,C 0.0069,E1 2.4021,E2 350.9508} C_DIS
LIN {X -34.0934,Y 135.9604,Z 187,A 104.4456,B 2.4326,C 0.0087,E1 2.398,E2 349.4493} C_DIS
LIN {X -38.7775,Y 134.7001,Z 187,A 106.7056,B 2.4326,C 0.0086,E1 2.3919,E2 347.1563} C_DIS
LIN {X -42.3358,Y 133.6233,Z 187,A 108.1036,B 2.4326,C 0.0102,E1 2.3882,E2 345.7741} C_DIS
LIN {X -46.2521,Y 132.3188,Z 187,A 110.5045,B 2.4326,C 0.0083,E1 2.3816,E2 343.2857} C_DIS
LIN {X -51.0181,Y 130.555,Z 187,A 111.7698,B 2.4326,C 0.0136,E1 2.3786,E2 342.1223} C_DIS
LIN {X -55.7024,Y 128.6259,Z 187,A 114.1021,B 2.4326,C 0.0144,E1 2.3725,E2 339.7591} C_DIS
LIN {X -58.5575,Y 127.3518,Z 187,A 116.1466,B 2.4326,C 0.0126,E1 2.367,E2 337.6201} C_DIS
LIN {X -63.6322,Y 124.8932,Z 187,A 117.7706,B 2.4326,C 0.018,E1 2.3632,E2 336.0825} C_DIS
LIN {X -66.8759,Y 123.1894,Z 187,A 119.4228,B 2.4326,C 0.0191,E1 2.359,E2 334.4122} C_DIS
LIN {X -69.7403,Y 121.5908,Z 187,A 121.4642,B 2.4326,C 0.0182,E1 2.3539,E2 332.2842} C_DIS
LIN {X -74.7535,Y 118.5742,Z 187,A 123.1188,B 2.4326,C 0.0242,E1 2.3502,E2 330.7234} C_DIS
LIN {X -78.7065,Y 115.9881,Z 187,A 125.1872,B 2.4325,C 0.0265,E1 2.3453,E2 328.6392} C_DIS
LIN {X -81.6986,Y 113.9005,Z 187,A 126.6855,B 2.4325,C 0.0287,E1 2.3419,E2 327.141} C_DIS
LIN {X -85.7089,Y 110.9142,Z 187,A 128.9038,B 2.4325,C 0.0313,E1 2.3369,E2 324.9024} C_DIS
LIN {X -88.7366,Y 108.5069,Z 187,A 130.5027,B 2.4324,C 0.0339,E1 2.3334,E2 323.3025} C_DIS
LIN {X -92.1108,Y 105.6576,Z 187,A 132.1905,B 2.4324,C 0.0374,E1 2.3299,E2 321.6306} C_DIS
LIN {X -94.0429,Y 103.9418,Z 187,A 133.6572,B 2.4324,C 0.0379,E1 2.3267,E2 320.1133} C_DIS
LIN {X -97.8591,Y 100.3578,Z 187,A 135.7538,B 2.4323,C 0.0421,E1 2.3225,E2 318.0238} C_DIS
LIN {X -100.9746,Y 97.2224,Z 187,A 137.6188,B 2.4323,C 0.0454,E1 2.3189,E2 316.1528} C_DIS
LIN {X -103.2526,Y 94.7989,Z 187,A 139.6432,B 2.4322,C 0.046,E1 2.3149,E2 314.0453} C_DIS
LIN {X -106.8627,Y 90.71,Z 187,A 141.1767,B 2.4321,C 0.0527,E1 2.3123,E2 312.6015} C_DIS
LIN {X -109.8528,Y 87.0653,Z 187,A 143.3576,B 2.432,C 0.0561,E1 2.3084,E2 310.3901} C_DIS
LIN {X -112.1233,Y 84.1216,Z 187,A 145.0624,B 2.432,C 0.0588,E1 2.3055,E2 308.6631} C_DIS
LIN {X -114.6328,Y 80.6677,Z 187,A 147.0132,B 2.4318,C 0.0622,E1 2.3023,E2 306.6875} C_DIS
LIN {X -116.5207,Y 77.9158,Z 187,A 148.6936,B 2.4318,C 0.0644,E1 2.2996,E2 304.9678} C_DIS
LIN {X -119.0299,Y 74.0257,Z 187,A 150.2174,B 2.4316,C 0.0698,E1 2.2974,E2 303.4924} C_DIS
LIN {X -121.0536,Y 70.6689,Z 187,A 151.8639,B 2.4316,C 0.0735,E1 2.2951,E2 301.8414} C_DIS
LIN {X -123.1824,Y 66.8887,Z 187,A 153.7466,B 2.4314,C 0.0775,E1 2.2925,E2 299.9461} C_DIS
LIN {X -124.9254,Y 63.5688,Z 187,A 155.3139,B 2.4313,C 0.0812,E1 2.2905,E2 298.3755} C_DIS
LIN {X -126.4345,Y 60.5119,Z 187,A 156.7963,B 2.4312,C 0.0845,E1 2.2887,E2 296.8828} C_DIS
LIN {X -127.9391,Y 57.2622,Z 187,A 158.1735,B 2.431,C 0.0884,E1 2.2871,E2 295.5177} C_DIS
LIN {X -129.2382,Y 54.2673,Z 187,A 159.7543,B 2.431,C 0.0912,E1 2.2853,E2 293.9064} C_DIS
LIN {X -130.5513,Y 51.0276,Z 187,A 161.2697,B 2.4308,C 0.0947,E1 2.2837,E2 292.381} C_DIS
LIN {X -131.7781,Y 47.77,Z 187,A 162.6466,B 2.4306,C 0.0985,E1 2.2824,E2 291.0111} C_DIS
LIN {X -132.7206,Y 45.0929,Z 187,A 164.0636,B 2.4306,C 0.101,E1 2.2811,E2 289.562} C_DIS
LIN {X -133.9391,Y 41.3259,Z 187,A 165.6714,B 2.4304,C 0.1053,E1 2.2797,E2 287.9566} C_DIS
LIN {X -134.9735,Y 37.8098,Z 187,A 167.2199,B 2.4302,C 0.1092,E1 2.2785,E2 286.4027} C_DIS
LIN {X -135.86,Y 34.4891,Z 187,A 168.7653,B 2.43,C 0.1127,E1 2.2774,E2 284.8403} C_DIS
LIN {X -136.535,Y 31.716,Z 187,A 170.4083,B 2.43,C 0.1147,E1 2.2764,E2 283.1364} C_DIS
LIN {X -137.3358,Y 28.0417,Z 187,A 171.6036,B 2.4297,C 0.1198,E1 2.2757,E2 281.9865} C_DIS
LIN {X -138.0023,Y 24.553,Z 187,A 173.1514,B 2.4295,C 0.1235,E1 2.2749,E2 280.4273} C_DIS
LIN {X -138.98,Y 18.2219,Z 187,A 175.9345,B 2.4291,C 0.1304,E1 2.2738,E2 277.6247} C_DIS
LIN {X -139.6601,Y 11.9404,Z 187,A 178.7097,B 2.4288,C 0.1372,E1 2.273,E2 274.8262} C_DIS
LIN {X -140.1171,Y 3.838,Z 187,A -177.8341,B 2.4282,C 0.1462,E1 2.2725,E2 271.3542} C_DIS
LIN {X -140.1636,Y -1.4969,Z 187,A -175.3436,B 2.4279,C 0.1516,E1 2.2725,E2 268.8245} C_DIS
LIN {X -140.0882,Y -4.821,Z 187,A -173.0249,B 2.4279,C 0.153,E1 2.2728,E2 266.3795} C_DIS
LIN {X -139.6904,Y -11.5815,Z 187,A -171.2465,B 2.4272,C 0.1632,E1 2.2731,E2 264.7341} C_DIS
LIN {X -139.1465,Y -16.9065,Z 187,A -168.6867,B 2.4268,C 0.1684,E1 2.2739,E2 262.1265} C_DIS
LIN {X -138.7342,Y -20.0083,Z 187,A -166.6425,B 2.4267,C 0.17,E1 2.2747,E2 259.9812} C_DIS
LIN {X -137.8132,Y -25.603,Z 187,A -164.799,B 2.4261,C 0.1776,E1 2.2756,E2 258.2024} C_DIS
LIN {X -137.0294,Y -29.5022,Z 187,A -163.2142,B 2.4258,C 0.1822,E1 2.2765,E2 256.6238} C_DIS
LIN {X -136.3087,Y -32.6712,Z 187,A -161.7904,B 2.4256,C 0.1855,E1 2.2774,E2 255.1881} C_DIS
LIN {X -135.4674,Y -36.0003,Z 187,A -160.3153,B 2.4253,C 0.1891,E1 2.2785,E2 253.704} C_DIS
LIN {X -134.4703,Y -39.5625,Z 187,A -158.7225,B 2.425,C 0.193,E1 2.2797,E2 252.1012} C_DIS
LIN {X -133.4995,Y -42.7235,Z 187,A -157.2281,B 2.4247,C 0.1962,E1 2.281,E2 250.5883} C_DIS
LIN {X -132.1643,Y -46.6977,Z 187,A -155.1494,B 2.4244,C 0.1997,E1 2.2829,E2 248.4615} C_DIS
LIN {X -131.0526,Y -49.7288,Z 187,A -153.7973,B 2.4242,C 0.203,E1 2.2843,E2 247.1055} C_DIS
LIN {X -129.392,Y -53.8991,Z 187,A -152.2025,B 2.4237,C 0.2084,E1 2.2859,E2 245.5438} C_DIS
LIN {X -127.9514,Y -57.2346,Z 187,A -150.5501,B 2.4234,C 0.2117,E1 2.2878,E2 243.8695} C_DIS
LIN {X -126.4697,Y -60.4381,Z 187,A -149.0516,B 2.4231,C 0.2151,E1 2.2896,E2 242.364} C_DIS
LIN {X -125.0162,Y -63.3906,Z 187,A -147.8019,B 2.4228,C 0.2187,E1 2.2911,E2 241.1277} C_DIS
LIN {X -123.5815,Y -66.1482,Z 187,A -146.0871,B 2.4226,C 0.2205,E1 2.2934,E2 239.3534} C_DIS
LIN {X -120.6016,Y -71.4377,Z 187,A -143.5252,B 2.4221,C 0.2261,E1 2.297,E2 236.7814} C_DIS
LIN {X -118.6455,Y -74.6405,Z 187,A -141.933,B 2.4218,C 0.2295,E1 2.2994,E2 235.1817} C_DIS
LIN {X -116.0822,Y -78.5675,Z 187,A -139.9458,B 2.4214,C 0.2336,E1 2.3025,E2 233.1856} C_DIS
LIN {X -113.3879,Y -82.4084,Z 187,A -136.9264,B 2.4214,C 0.2342,E1 2.3077,E2 230.0153} C_DIS
LIN {X -108.7887,Y -88.3917,Z 187,A -134.6601,B 2.4204,C 0.2434,E1 2.3114,E2 227.8625} C_DIS
LIN {X -106.6716,Y -90.9348,Z 187,A -132.9891,B 2.4203,C 0.2451,E1 2.3146,E2 226.1482} C_DIS
LIN {X -104.1329,Y -93.832,Z 187,A -131.625,B 2.4199,C 0.249,E1 2.317,E2 224.8133} C_DIS
LIN {X -101.0671,Y -97.1263,Z 187,A -129.7117,B 2.4195,C 0.2522,E1 2.3207,E2 222.8901} C_DIS
LIN {X -94.8051,Y -103.2469,Z 187,A -126.0038,B 2.4189,C 0.2583,E1 2.3282,E2 219.1651} C_DIS
LIN {X -90.4954,Y -107.0451,Z 187,A -123.544,B 2.4185,C 0.2619,E1 2.3335,E2 216.69} C_DIS
LIN {X -86.9519,Y -109.9431,Z 187,A -121.5942,B 2.4182,C 0.2646,E1 2.3377,E2 214.7294} C_DIS
LIN {X -82.6564,Y -113.2077,Z 187,A -119.0235,B 2.418,C 0.2665,E1 2.3436,E2 212.1081} C_DIS
LIN {X -79.4083,Y -115.5087,Z 187,A -117.6776,B 2.4176,C 0.27,E1 2.3466,E2 210.8012} C_DIS
LIN {X -76.216,Y -117.6395,Z 187,A -116.0614,B 2.4174,C 0.272,E1 2.3504,E2 209.1783} C_DIS
LIN {X -72.2458,Y -120.1191,Z 187,A -114.0911,B 2.4171,C 0.2743,E1 2.3552,E2 207.2} C_DIS
LIN {X -68.3281,Y -122.3902,Z 187,A -112.3134,B 2.4168,C 0.2769,E1 2.3595,E2 205.4323} C_DIS
LIN {X -65.3325,Y -124.0123,Z 187,A -110.4878,B 2.4168,C 0.2765,E1 2.3641,E2 203.5463} C_DIS
LIN {X -62.0033,Y -125.7098,Z 187,A -109.3362,B 2.4165,C 0.2799,E1 2.3669,E2 202.4468} C_DIS
LIN {X -59.1825,Y -127.0628,Z 187,A -108.1398,B 2.4163,C 0.2816,E1 2.3699,E2 201.2617} C_DIS
LIN {X -55.9238,Y -128.5302,Z 187,A -106.6142,B 2.4162,C 0.2827,E1 2.3738,E2 199.7269} C_DIS
LIN {X -52.6175,Y -129.9186,Z 187,A -104.9443,B 2.4162,C 0.283,E1 2.3782,E2 198.0283} C_DIS
LIN {X -49.2079,Y -131.2477,Z 187,A -102.7834,B 2.4164,C 0.2809,E1 2.3841,E2 195.7741} C_DIS
LIN {X -43.9417,Y -133.1039,Z 187,A -101.0859,B 2.4158,C 0.2855,E1 2.3884,E2 194.1579} C_DIS
LIN {X -39.7664,Y -134.4106,Z 187,A -99.3599,B 2.4157,C 0.2869,E1 2.393,E2 192.4402} C_DIS
LIN {X -33.5091,Y -136.1067,Z 187,A -96.4571,B 2.4157,C 0.2869,E1 2.4009,E2 189.5014} C_DIS
LIN {X -28.4068,Y -137.2615,Z 187,A -94.4571,B 2.4155,C 0.2885,E1 2.4063,E2 187.52} C_DIS
LIN {X -23.9143,Y -138.1166,Z 187,A -92.4978,B 2.4155,C 0.2886,E1 2.4118,E2 185.5475} C_DIS
LIN {X -20.1359,Y -138.7159,Z 187,A -90.9866,B 2.4154,C 0.2892,E1 2.4159,E2 184.0431} C_DIS
LIN {X -16.1328,Y -139.2388,Z 187,A -89.3162,B 2.4154,C 0.2894,E1 2.4206,E2 182.3691} C_DIS
LIN {X -11.8647,Y -139.6665,Z 187,A -87.6246,B 2.4154,C 0.2898,E1 2.4253,E2 180.6854} C_DIS
LIN {X -8.0488,Y -139.9394,Z 187,A -86.0966,B 2.4153,C 0.29,E1 2.4295,E2 179.1617} C_DIS
LIN {X -4.4883,Y -140.099,Z 187,A -84.5359,B 2.4153,C 0.2892,E1 2.4339,E2 177.5859} C_DIS
LIN {X -0.3093,Y -140.1701,Z 187,A -82.8792,B 2.4153,C 0.2892,E1 2.4386,E2 175.9356} C_DIS
LIN {X -0.3093,Y -140.1701,Z 187,A -82.8792,B 2.4153,C 0.2892,E1 2.4386,E2 175.9356} C_DIS
Enddeposition()
LIN {X 0.9952,Y -141.0634,Z 187,A -82.8975,B 2.4277,C 0.2943,E1 2.4511,E2 176.0566} C_DIS
Startdeposition()
$VEL.CP = VEL_PRINT
LIN {X -2.4561,Y -141.048,Z 187,A -84.4341,B 2.4276,C 0.2954,E1 2.4467,E2 177.6128} C_DIS
LIN {X -6.314,Y -140.93,Z 187,A -86.1357,B 2.4275,C 0.2963,E1 2.4419,E2 179.3337} C_DIS
LIN {X -10.3468,Y -140.6893,Z 187,A -87.6189,B 2.4275,C 0.2954,E1 2.4378,E2 180.7957} C_DIS
LIN {X -14.0813,Y -140.3659,Z 187,A -89.1605,B 2.4275,C 0.2954,E1 2.4335,E2 182.3406} C_DIS
LIN {X -18.1159,Y -139.9013,Z 187,A -90.8126,B 2.4275,C 0.2952,E1 2.4289,E2 183.9937} C_DIS
LIN {X -21.581,Y -139.4086,Z 187,A -92.2471,B 2.4276,C 0.295,E1 2.425,E2 185.4306} C_DIS
LIN {X -25.4074,Y -138.7633,Z 187,A -93.7705,B 2.4277,C 0.2943,E1 2.4208,E2 186.9472} C_DIS
LIN {X -28.2827,Y -138.2049,Z 187,A -95.0365,B 2.4277,C 0.2943,E1 2.4173,E2 188.2243} C_DIS
LIN {X -32.2454,Y -137.3366,Z 187,A -96.654,B 2.4278,C 0.2934,E1 2.4129,E2 189.8381} C_DIS
LIN {X -35.6912,Y -136.4808,Z 187,A -98.1371,B 2.4278,C 0.2929,E1 2.4088,E2 191.3274} C_DIS
LIN {X -39.2519,Y -135.4987,Z 187,A -99.4781,B 2.4281,C 0.2912,E1 2.4053,E2 192.6467} C_DIS
LIN {X -42.1635,Y -134.6229,Z 187,A -101.3154,B 2.4278,C 0.2935,E1 2.4001,E2 194.5678} C_DIS
LIN {X -45.8311,Y -133.4162,Z 187,A -102.6654,B 2.4281,C 0.2913,E1 2.3966,E2 195.8881} C_DIS
LIN {X -49.9452,Y -131.9323,Z 187,A -104.2875,B 2.4283,C 0.2891,E1 2.3924,E2 197.4892} C_DIS
LIN {X -53.4468,Y -130.5543,Z 187,A -105.9393,B 2.4284,C 0.2884,E1 2.3881,E2 199.1584} C_DIS
LIN {X -58.0001,Y -128.5946,Z 187,A -107.9051,B 2.4287,C 0.2863,E1 2.3831,E2 201.1179} C_DIS
LIN {X -61.2412,Y -127.0832,Z 187,A -109.3956,B 2.4288,C 0.285,E1 2.3793,E2 202.614} C_DIS
LIN {X -64.7278,Y -125.3449,Z 187,A -111.3647,B 2.4288,C 0.285,E1 2.3743,E2 204.6367} C_DIS
LIN {X -67.9918,Y -123.6051,Z 187,A -112.5648,B 2.4292,C 0.2819,E1 2.3714,E2 205.7954} C_DIS
LIN {X -71.6813,Y -121.5023,Z 187,A -114.4165,B 2.4294,C 0.2803,E1 2.3669,E2 207.6647} C_DIS
LIN {X -75.3622,Y -119.2539,Z 187,A -116.0678,B 2.4297,C 0.2775,E1 2.363,E2 209.3023} C_DIS
LIN {X -78.5341,Y -117.1896,Z 187,A -117.7742,B 2.4298,C 0.2761,E1 2.359,E2 211.032} C_DIS
LIN {X -82.1369,Y -114.6931,Z 187,A -120.0428,B 2.4299,C 0.2755,E1 2.3536,E2 213.3677} C_DIS
LIN {X -85.7164,Y -112.0431,Z 187,A -121.4796,B 2.4304,C 0.2712,E1 2.3506,E2 214.7535} C_DIS
LIN {X -89.2356,Y -109.261,Z 187,A -123.3895,B 2.4307,C 0.2686,E1 2.3464,E2 216.6754} C_DIS
LIN {X -93.7379,Y -105.4245,Z 187,A -125.7781,B 2.4311,C 0.2644,E1 2.3413,E2 219.062} C_DIS
LIN {X -99.6338,Y -99.8706,Z 187,A -128.9472,B 2.4318,C 0.258,E1 2.3349,E2 222.2143} C_DIS
LIN {X -102.8841,Y -96.5192,Z 187,A -131.1102,B 2.4321,C 0.2554,E1 2.3306,E2 224.4137} C_DIS
LIN {X -105.336,Y -93.8372,Z 187,A -133.1953,B 2.4321,C 0.2546,E1 2.3266,E2 226.5814} C_DIS
LIN {X -108.1099,Y -90.6267,Z 187,A -134.5796,B 2.4327,C 0.2499,E1 2.3242,E2 227.9195} C_DIS
LIN {X -114.1885,Y -82.8368,Z 187,A -138.7401,B 2.4335,C 0.2418,E1 2.3171,E2 232.0992} C_DIS
LIN {X -116.5925,Y -79.4186,Z 187,A -140.6252,B 2.4338,C 0.2386,E1 2.314,E2 234.0093} C_DIS
LIN {X -119.2201,Y -75.4158,Z 187,A -142.6036,B 2.4342,C 0.2343,E1 2.311,E2 235.9917} C_DIS
LIN {X -121.4826,Y -71.7148,Z 187,A -144.5195,B 2.4346,C 0.2306,E1 2.3082,E2 237.9278} C_DIS
LIN {X -124.5252,Y -66.2909,Z 187,A -147.0269,B 2.4351,C 0.2245,E1 2.3049,E2 240.4319} C_DIS
LIN {X -125.8449,Y -63.7458,Z 187,A -148.306,B 2.4354,C 0.222,E1 2.3032,E2 241.726} C_DIS
LIN {X -127.4321,Y -60.5107,Z 187,A -149.9064,B 2.4357,C 0.2188,E1 2.3012,E2 243.3442} C_DIS
LIN {X -129.3112,Y -56.3845,Z 187,A -151.6033,B 2.4361,C 0.2137,E1 2.2993,E2 245.021} C_DIS
LIN {X -130.9645,Y -52.4292,Z 187,A -153.6114,B 2.4364,C 0.21,E1 2.2971,E2 247.0642} C_DIS
LIN {X -133.0131,Y -46.9959,Z 187,A -156.2354,B 2.4369,C 0.2046,E1 2.2946,E2 249.7228} C_DIS
LIN {X -134.4042,Y -42.8481,Z 187,A -157.9543,B 2.4373,C 0.1997,E1 2.2931,E2 251.433} C_DIS
LIN {X -135.4079,Y -39.5619,Z 187,A -159.4775,B 2.4376,C 0.1964,E1 2.2918,E2 252.9726} C_DIS
LIN {X -136.4023,Y -35.9861,Z 187,A -161.0294,B 2.4379,C 0.1924,E1 2.2907,E2 254.5297} C_DIS
LIN {X -137.1477,Y -33.0296,Z 187,A -162.3567,B 2.4381,C 0.1893,E1 2.2898,E2 255.8682} C_DIS
LIN {X -137.9255,Y -29.6152,Z 187,A -163.9381,B 2.4384,C 0.1858,E1 2.2888,E2 257.4699} C_DIS
LIN {X -138.6953,Y -25.78,Z 187,A -166.5303,B 2.4385,C 0.184,E1 2.2875,E2 260.193} C_DIS
LIN {X -139.7751,Y -19.0789,Z 187,A -169.5761,B 2.4391,C 0.177,E1 2.2863,E2 263.2747} C_DIS
LIN {X -140.5743,Y -11.8065,Z 187,A -171.6347,B 2.4398,C 0.1665,E1 2.2858,E2 265.2125} C_DIS
LIN {X -140.9525,Y -5.7446,Z 187,A -174.0655,B 2.4403,C 0.1595,E1 2.2854,E2 267.6373} C_DIS
LIN {X -141.0471,Y -2.5099,Z 187,A -175.6863,B 2.4405,C 0.1566,E1 2.2853,E2 269.2974} C_DIS
LIN {X -141.0632,Y 1.5044,Z 187,A -177.7285,B 2.4407,C 0.153,E1 2.2853,E2 271.3923} C_DIS
LIN {X -140.9852,Y 4.9027,Z 187,A -179.3342,B 2.4409,C 0.1496,E1 2.2855,E2 273.0263} C_DIS
LIN {X -140.7793,Y 9.0483,Z 187,A 179.4088,B 2.4412,C 0.1439,E1 2.2857,E2 274.2265} C_DIS
LIN {X -140.5478,Y 12.12,Z 187,A 178.0333,B 2.4414,C 0.1407,E1 2.286,E2 275.6174} C_DIS
LIN {X -140.2538,Y 15.1455,Z 187,A 176.6779,B 2.4416,C 0.1375,E1 2.2864,E2 276.9876} C_DIS
LIN {X -139.7921,Y 18.9487,Z 187,A 174.4511,B 2.4418,C 0.1348,E1 2.2873,E2 279.2999} C_DIS
LIN {X -139.0575,Y 23.7438,Z 187,A 172.862,B 2.4421,C 0.1284,E1 2.2879,E2 280.8387} C_DIS
LIN {X -138.0058,Y 29.2405,Z 187,A 170.3865,B 2.4424,C 0.1226,E1 2.2893,E2 283.3386} C_DIS
LIN {X -137.0238,Y 33.5439,Z 187,A 168.6215,B 2.4426,C 0.1177,E1 2.2904,E2 285.0989} C_DIS
LIN {X -135.9199,Y 37.7662,Z 187,A 166.7027,B 2.4428,C 0.1132,E1 2.2918,E2 287.0351} C_DIS
LIN {X -134.945,Y 41.1135,Z 187,A 165.22,B 2.443,C 0.1096,E1 2.293,E2 288.5254} C_DIS
LIN {X -133.7917,Y 44.724,Z 187,A 163.6294,B 2.4432,C 0.1056,E1 2.2944,E2 290.1214} C_DIS
LIN {X -132.5715,Y 48.2221,Z 187,A 162.0459,B 2.4433,C 0.1019,E1 2.2959,E2 291.7139} C_DIS
LIN {X -131.3397,Y 51.4825,Z 187,A 160.5343,B 2.4435,C 0.0984,E1 2.2974,E2 293.2367} C_DIS
LIN {X -130.0155,Y 54.7407,Z 187,A 159.036,B 2.4436,C 0.0949,E1 2.299,E2 294.7429} C_DIS
LIN {X -128.4833,Y 58.249,Z 187,A 157.3707,B 2.4438,C 0.0913,E1 2.3009,E2 296.4211} C_DIS
LIN {X -127.1458,Y 61.1101,Z 187,A 156.0369,B 2.4438,C 0.0882,E1 2.3026,E2 297.7604} C_DIS
LIN {X -125.4954,Y 64.4323,Z 187,A 154.4239,B 2.444,C 0.0847,E1 2.3046,E2 299.3858} C_DIS
LIN {X -123.2219,Y 68.684,Z 187,A 152.3281,B 2.4441,C 0.0803,E1 2.3074,E2 301.4976} C_DIS
LIN {X -121.0547,Y 72.4347,Z 187,A 150.4764,B 2.4443,C 0.0764,E1 2.3101,E2 303.3596} C_DIS
LIN {X -118.7343,Y 76.1784,Z 187,A 148.4095,B 2.4443,C 0.073,E1 2.3132,E2 305.4601} C_DIS
LIN {X -115.7918,Y 80.5806,Z 187,A 146.6112,B 2.4445,C 0.0671,E1 2.3159,E2 307.2125} C_DIS
LIN {X -113.6613,Y 83.5587,Z 187,A 144.9232,B 2.4446,C 0.0643,E1 2.3187,E2 308.9248} C_DIS
LIN {X -111.9264,Y 85.869,Z 187,A 143.5252,B 2.4446,C 0.0624,E1 2.3211,E2 310.3501} C_DIS
LIN {X -108.8659,Y 89.7178,Z 187,A 141.6196,B 2.4448,C 0.0579,E1 2.3245,E2 312.2427} C_DIS
LIN {X -106.6566,Y 92.3334,Z 187,A 139.5186,B 2.4448,C 0.0572,E1 2.3285,E2 314.4312} C_DIS
LIN {X -103.5629,Y 95.7907,Z 187,A 138.0511,B 2.4449,C 0.0522,E1 2.3311,E2 315.8456} C_DIS
LIN {X -100.5508,Y 98.9472,Z 187,A 136.1814,B 2.4449,C 0.049,E1 2.3348,E2 317.7261} C_DIS
LIN {X -97.3969,Y 102.0529,Z 187,A 134.3152,B 2.445,C 0.0459,E1 2.3385,E2 319.5996} C_DIS
Enddeposition()
END
